(* Logix 5000 project; controller CarbonScout_MK6 vendor 1 type 14 code 154 rev 32.11; software revision 32.00; part 4 of 17 *)
(* tags used below, declared in another part *)
   Cfg_Exists : BOOL;   // 1=Alarm configured to exist, 0=Does not exist, don't scan
   Cfg_ResetReqd : BOOL;   // 1=Latched Alarm, a Reset is required to clear this Alarm
   Cfg_AckReqd : BOOL;   // 1=Acknowledge required for this Alarm
   Cfg_AllowShelve : BOOL;   // 1=Allow Operator to Shelve this Alarm
   Cfg_AllowDisable : BOOL;   // 1=Allow Maintenance to Disable this Alarm
   Cfg_Severity : DINT;   // Alarm Severity: 1..250=Low, 251..500=Medium, 501..750=High, 751..1000=Urgent
   Cfg_AlmMinOnT : DINT;   // Minimum time Alm output stays on (sec)
   PCfg_AllowExist : BOOL;   // 1=Alarm can be configured to exist, 0=other configs make alarm meaningless
   PCmd_Ack : BOOL;   // Program Command to Acknowledge alarm
   PCmd_Suppress : BOOL;   // Program Command to Suppress by Design (inhibits new alarm)
   PCmd_Unsuppress : BOOL;   // Program Command to Unsuppress (allows new alarm)
   PCmd_Unshelve : BOOL;   // Program Command to Unshelve (e.g., on shift change)
   OCmd_Ack : BOOL;   // Operator Command to Acknowledge alarm
   OCmd_Shelve : BOOL;   // Operator Command to Shelve Alarm (inhibits new alarm)
   OCmd_Unshelve : BOOL;   // Operator Command to Unshelve alarm (allows new alarm)
   Alm : ALIAS FOR Com_AE.0;   // Alarm output 1=In Alarm
   Ack : ALIAS FOR Com_AE.1;   // Alarm acknowledged status: 1=Ack rcvd
   Shelved : ALIAS FOR Com_AE.3;   // 1=Alarm has been Shelved by Operator (inhibits new alarm)
   Suppressed : ALIAS FOR Com_AE.6;   // 1=Alarm has been Suppressed by Program (inhibits new alarm)
   Disabled : ALIAS FOR Com_AE.9;   // 1=Alarm has been Disabled by Maintanance (inhibits new alarm)
   P_Alarm : BOOL;   // Unique Parameter Name for auto - discovery
   Wrk_Suppressed : BOOL;   // Internal Alarm Suppressed Status
   Com_AE : DINT;   // Communication with HMI / Alarm/Event Server (see bit descriptions)
   Simulation : DINT;
   test : DINT;
(* P_Alarm, continued *)

ROUTINE Prescan   (* ladder *)
// Clear "lurking" Commands
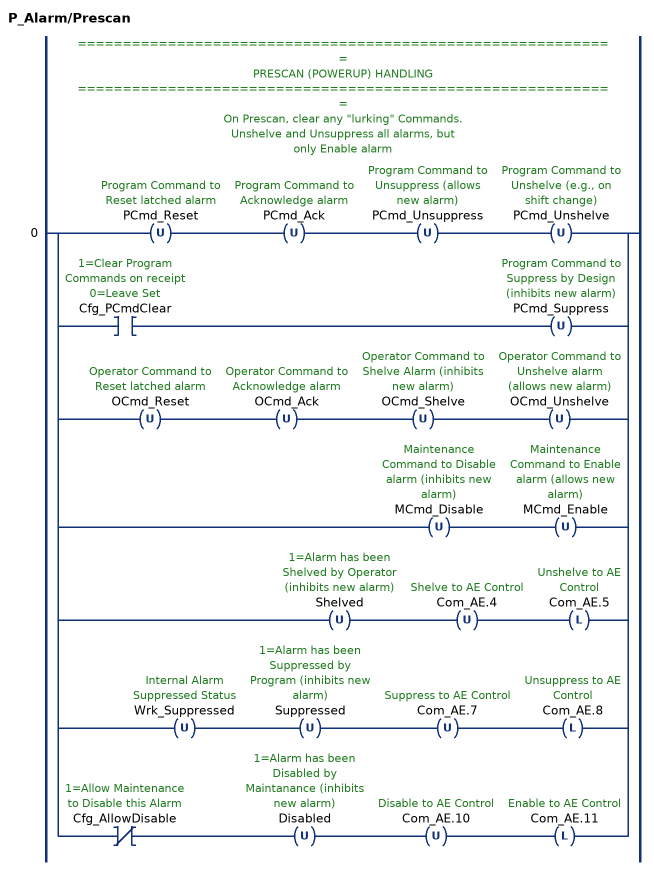
   // ============================================================
   // PRESCAN (POWERUP) HANDLING
   // ============================================================
   // On Prescan, clear any "lurking" Commands.
   // Unshelve and Unsuppress all alarms, but
   // only Enable alarm
   0: [OTU(PCmd_Reset) OTU(PCmd_Ack) OTU(PCmd_Unsuppress) OTU(PCmd_Unshelve) ,XIC(Cfg_PCmdClear) OTU(PCmd_Suppress) ,OTU(OCmd_Reset) OTU(OCmd_Ack) OTU(OCmd_Shelve) OTU(OCmd_Unshelve) ,OTU(MCmd_Disable) OTU(MCmd_Enable) ,OTU(Shelved) OTU(Com_AE.4) OTL(Com_AE.5) ,OTU(Wrk_Suppressed) OTU(Suppressed) OTU(Com_AE.7) OTL(Com_AE.8) ,XIO(Cfg_AllowDisable) OTU(Disabled) OTU(Com_AE.10) OTL(Com_AE.11) ];
END_ROUTINE
END_ADD_ON_INSTRUCTION

ADD_ON_INSTRUCTION P_Gate   (* revision 3.5 01 Release, vendor Rockwell Automation, ExecutePrescan, ExecuteEnableInFalse *)
// Condition Gate/Delay
// Revision note:
// See V3.5-xx Release Notes for details. Unchanged, up-rev only for V3.5 Library.
// Help:
// Copyright © Rockwell Automation, Inc.  All Rights Reserved.
// This Instruction provides a "gate" for a discrete Input signal and
// provides on-delay and off-delay timing for the gated signal.
// When the Gate input is true, the instruction Input is passed through
// to the Output, with on-delay and off-delay timing applied.
// When the Gate input is false, the Output is kept off
// (note: off-delay still applies!)
// This instruction is usually used between a comparison
// (analog threshold with deadband or discrete logic)
// and a P_Alarm instance, but may be used as a
// gated on-delay/off-delay timer generally.
// When EnableIn  is FALSE (e.g., on a false LD rung),
// the Input "Inp" is inverted.  Note that the Gate
// input (Inp_Gate) is NOT inverted!!!
VAR_INPUT
   Inp : BOOL; {visible}   // Input Condition: e.g., result of comparison
   Inp_Gate : BOOL := 1; {visible}   // Gate Input: 1=enable On Delay / Off Delay after Gate Delay, 0=disable
   Cfg_GateDly : DINT;   // Gate Delay (s): time after Gate Input true to enable On/Off Delay
   Cfg_OnDly : DINT;   // On Delay (s): If Gate Delay done, time Inp must be true to set Out true
   Cfg_OffDly : DINT;   // Off Delay (s): Time after Inp or Gate goes to 0 for Out to go to 0
END_VAR
VAR_OUTPUT
   Out : BOOL; {access Read Only, visible}   // Output after On Delay, Off Delay, enabled by Gate
   Sts_Gate : BOOL; {access Read Only, visible}   // 1=Gate Delay done, Output is enabled
   Sts_Err : BOOL; {access Read Only, visible}   // 1=Error in Config (see detail Err_ bits for reason), display icon
   Err_Timer : BOOL; {access Read Only}   // 1=Error in Config: On Delay, Off Delay, Gate Delay Time Invalid (use 0 to 2147483 s)
   P_Gate : BOOL;   // Unique Parameter Name for auto - discovery
END_VAR
VAR
   Wrk_OffDlyT : TIMER; {access Read Only}   // Off Delay Timer
   Wrk_OnDlyT : TIMER; {access Read Only}   // On Delay Timer
   Wrk_GateT : TIMER; {access Read Only}   // Gate Delay Timer
   Cfg_InpCond : STRING_8;   // Displayed text of P_Gate's Input (Inp) Condition
   Inf_Tab : DINT;   // Tab to display (FTView ME)
END_VAR

ROUTINE EnableInFalse   (* ladder *)
// Same as main Logic routine, except Inp is inverted (for use in LD logic)  (Inp_Gate is NOT inverted!!!)
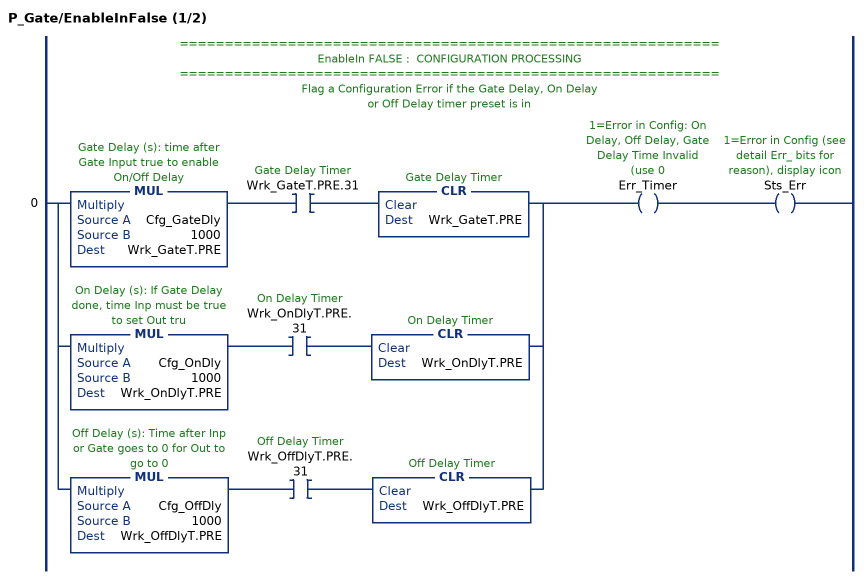
   // ============================================================
   // EnableIn FALSE :  CONFIGURATION PROCESSING
   // ============================================================
   // Flag a Configuration Error if the Gate Delay, On Delay
   // or Off Delay timer preset is in
   0: [MUL(Cfg_GateDly,1000,Wrk_GateT.PRE) XIC(Wrk_GateT.PRE.31) CLR(Wrk_GateT.PRE) ,MUL(Cfg_OnDly,1000,Wrk_OnDlyT.PRE) XIC(Wrk_OnDlyT.PRE.31) CLR(Wrk_OnDlyT.PRE) ,MUL(Cfg_OffDly,1000,Wrk_OffDlyT.PRE) XIC(Wrk_OffDlyT.PRE.31) CLR(Wrk_OffDlyT.PRE) ]OTE(Err_Timer)OTE(Sts_Err);
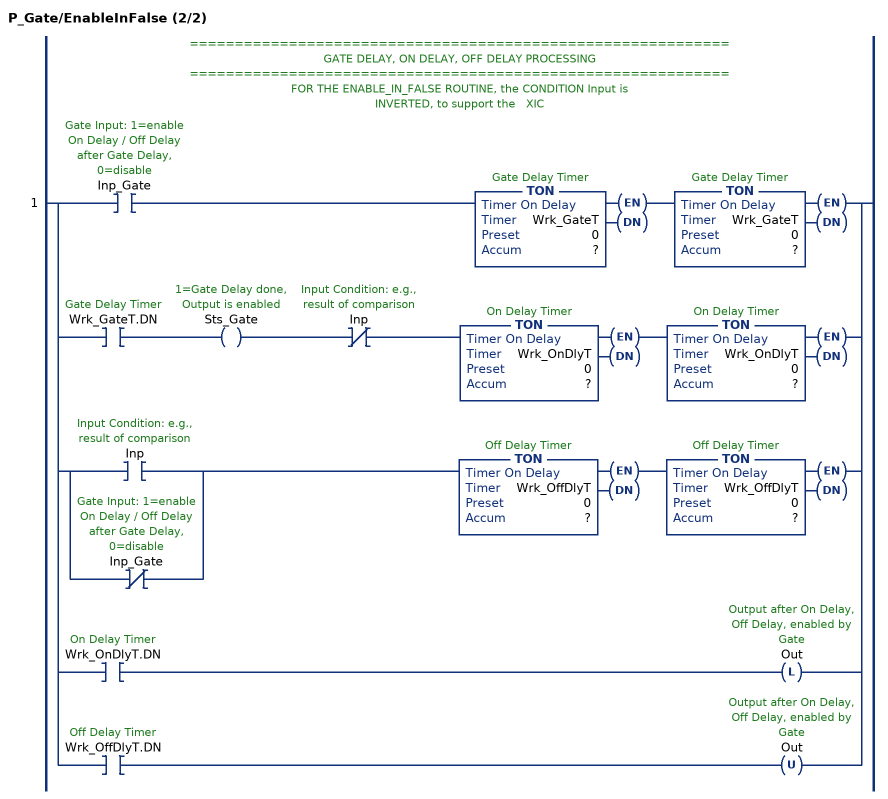
   // ============================================================
   // GATE DELAY, ON DELAY, OFF DELAY PROCESSING
   // ============================================================
   // FOR THE ENABLE_IN_FALSE ROUTINE, the CONDITION Input is
   // INVERTED, to support the   XIC
   1: [XIC(Inp_Gate) TON(Wrk_GateT,?,?) TON(Wrk_GateT,?,?) ,XIC(Wrk_GateT.DN) OTE(Sts_Gate) XIO(Inp) TON(Wrk_OnDlyT,?,?) TON(Wrk_OnDlyT,?,?) ,[XIC(Inp) ,XIO(Inp_Gate) ] TON(Wrk_OffDlyT,?,?) TON(Wrk_OffDlyT,?,?) ,XIC(Wrk_OnDlyT.DN) OTL(Out) ,XIC(Wrk_OffDlyT.DN) OTU(Out) ];
END_ROUTINE

ROUTINE Logic   (* ladder *)
// Gate the input and apply on-delay and off-delay timing
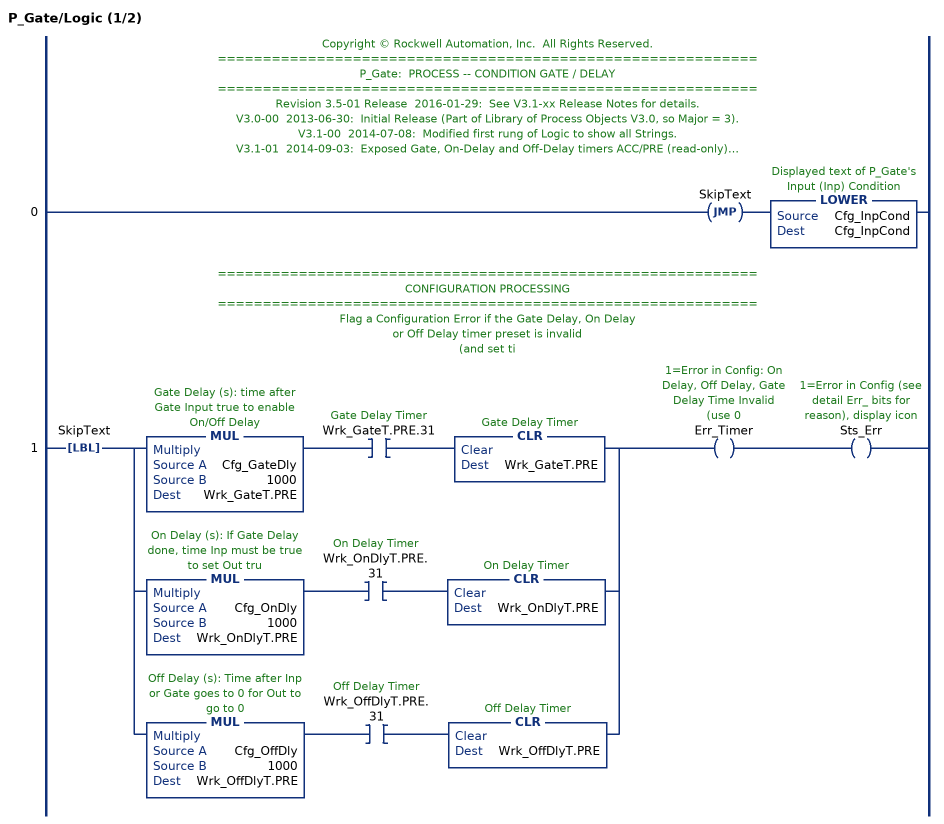
   // Copyright © Rockwell Automation, Inc.  All Rights Reserved.
   // ============================================================
   // P_Gate:  PROCESS -- CONDITION GATE / DELAY
   // ============================================================
   // Revision 3.5-01 Release  2016-01-29:  See V3.1-xx Release Notes for details.
   // V3.0-00  2013-06-30:  Initial Release (Part of Library of Process Objects V3.0, so Major = 3).
   // V3.1-00  2014-07-08:  Modified first rung of Logic to show all Strings.
   // V3.1-01  2014-09-03:  Exposed Gate, On-Delay and Off-Delay timers ACC/PRE (read-only).
   // V3.1-05  2016-01-22:  Corrected logic when using analog threshold with deadband.
   // V3.5-01  2016-01-29:  Unchanged, up-rev only for V3.5 Library.
   // ============================================================
   // This Instruction provides a "gate" for a discrete Input signal and
   // provides on-delay and off-delay timing for the gated signal.
   // When the Gate input is true, the instruction Input is passed through
   // to the Output, with on-delay and off-delay timing applied.
   // When the Gate input is false, the Output is kept off
   // (note: off-delay still applies!)
   // This instruction is usually used between a comparison
   // (analog threshold with deadband or discrete logic)
   // and a P_Alarm instance, but may be used as a
   // gated on-delay/off-delay timer generally.
   // When EnableIn  is FALSE (e.g., on a false LD rung),
   // the Input "Inp" is inverted.  Note that the Gate
   // input (Inp_Gate) is NOT inverted!!!
   // ============================================================
   // SHOW LOCAL STRINGS
   // ============================================================
   // The STRINGs containing the text associated with each instance of this
   // instruction cannot be Input or Output Parameters, because STRINGs are not
   //  'atomic' types. (Inputs and Outputs must be SINT, INT, DINT, REAL, or BOOL.)
   // In order to make it easier to find and configure these STRINGs, this rung
   // was added.  THE JMP (and the LBL on the following rung)
   // MUST NOT BE REMOVED!!!
   // To view the STRINGs, go to the instruction instance (in LD or FBD), RIGHT-click
   // to bring up the context menu and select "Open Instruction Logic".
   // This rung will appear with the STRING values for the selected instance.
   // You may double-click the STRING values here to modify them as well.
   // #####  V3.1-00  2014-07-08: Added Inf_Type to displayed Strings  #####
   0: JMP(SkipText)LOWER(Cfg_InpCond,Cfg_InpCond);
   // ============================================================
   // CONFIGURATION PROCESSING
   // ============================================================
   // Flag a Configuration Error if the Gate Delay, On Delay
   // or Off Delay timer preset is invalid
   // (and set ti
   1: LBL(SkipText)[MUL(Cfg_GateDly,1000,Wrk_GateT.PRE) XIC(Wrk_GateT.PRE.31) CLR(Wrk_GateT.PRE) ,MUL(Cfg_OnDly,1000,Wrk_OnDlyT.PRE) XIC(Wrk_OnDlyT.PRE.31) CLR(Wrk_OnDlyT.PRE) ,MUL(Cfg_OffDly,1000,Wrk_OffDlyT.PRE) XIC(Wrk_OffDlyT.PRE.31) CLR(Wrk_OffDlyT.PRE) ]OTE(Err_Timer)OTE(Sts_Err);
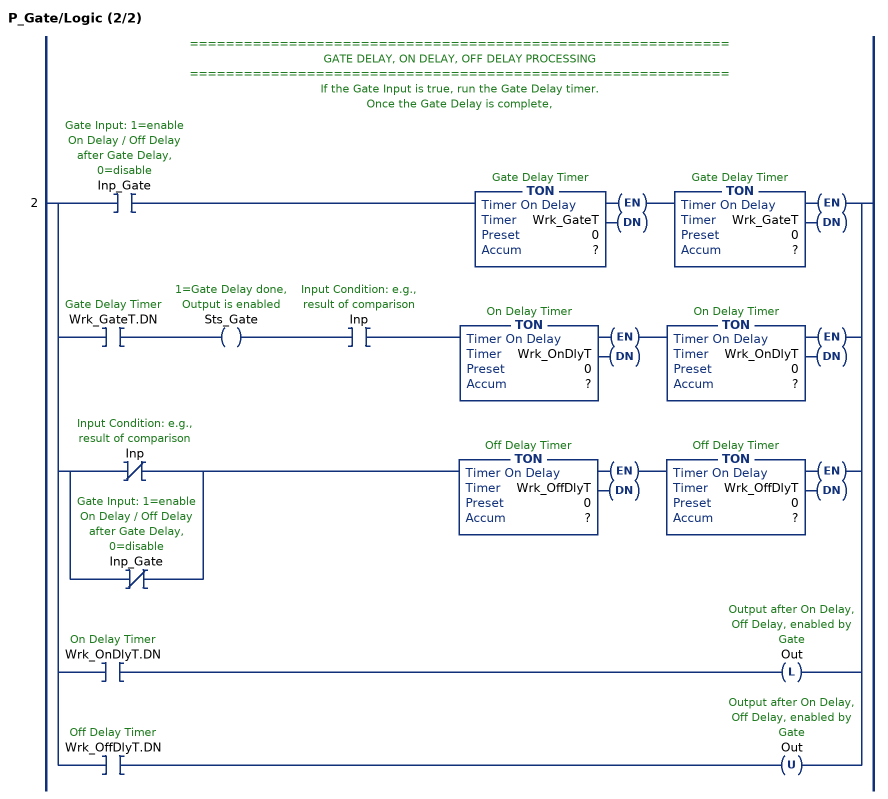
   // ============================================================
   // GATE DELAY, ON DELAY, OFF DELAY PROCESSING
   // ============================================================
   // If the Gate Input is true, run the Gate Delay timer.
   // Once the Gate Delay is complete,
   2: [XIC(Inp_Gate) TON(Wrk_GateT,?,?) TON(Wrk_GateT,?,?) ,XIC(Wrk_GateT.DN) OTE(Sts_Gate) XIC(Inp) TON(Wrk_OnDlyT,?,?) TON(Wrk_OnDlyT,?,?) ,[XIO(Inp) ,XIO(Inp_Gate) ] TON(Wrk_OffDlyT,?,?) TON(Wrk_OffDlyT,?,?) ,XIC(Wrk_OnDlyT.DN) OTL(Out) ,XIC(Wrk_OffDlyT.DN) OTU(Out) ];
END_ROUTINE

ROUTINE Prescan   (* ladder *)
// Set the Gate Input to 1 (default value) on prescan
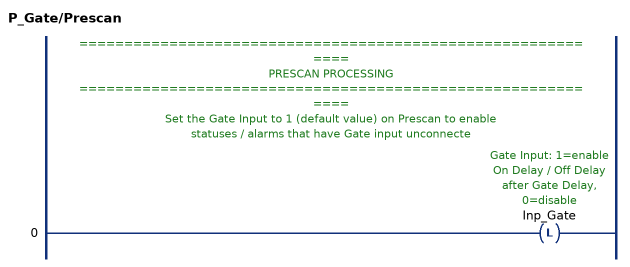
   // ============================================================
   // PRESCAN PROCESSING
   // ============================================================
   // Set the Gate Input to 1 (default value) on Prescan to enable
   // statuses / alarms that have Gate input unconnecte
   0: OTL(Inp_Gate);
END_ROUTINE
END_ADD_ON_INSTRUCTION

ADD_ON_INSTRUCTION P_Mode   (* revision 3.5 01 Release, vendor Rockwell Automation, ExecutePrescan, ExecuteEnableInFalse *)
// Mode
// Revision note:
// See V3.5-xx Release Notes for details. Unmodified, up-rev only for V3.5-01 Release.
// Help:
// Copyright © Rockwell Automation, Inc.  All Rights Reserved.
// This instruction provides selection of Mode (owner) for a Device level
// object  (from highest priority to lowest):
// *  No Mode (no owner, EnableIn is false)
// *  Hand (typically tracks hardwired control of device)
// *  Maint (Maintenance) (taken out of normal service for maintenance)
// *  Ovrd (Override) (typically used for process overrides)
// *  Prog  (Program) (automated control, and default if Cfg_ProgNorm = 1)
// *  Oper (Operator (manual control, and default if Cfg_ProgNorm = 0)
// (Program and Operator have the same priority.)
// The current mode is shown with Status bits and also as the primary
// Value for the instruction: an enumeration "Val" as follows:
//   0 = No Mode,
//   1 = Hand,
//   2 = Maintenance,
//   3 = Override,
//   4 = Program (Locked),
//   5 = Operator (Locked),
//   6 = Program (Unlocked, Oper default),
//   7 = Operator (Unlocked, Prog default),
//   8 = Program (Unlocked, = default),
//   9 = Operator (Unlocked, = default).
// When EnableIn is false, all ownership acquire/release and lock/unlock
// Commands are processed "behind the scenes", but the Mode is shown
// as "No Mode" (no owner).  When EnableIn becomes true, the Mode
// takes into account the Commands received -- in other words, the Mode
// becomes the one that would have been in effect had the EnableIn
// False / No Mode condition never occurred.
VAR_INPUT
   Inp_Hand : BOOL; {visible}   // 1=Acquire Hand (typ. hardwired local) Mode, 0=Release Hand Mode
   Inp_Ovrd : BOOL; {visible}   // 1=Acquire Override (higher priority program logic) Mode, 0=Release Override Mode
   Cfg_PCmdClear : BOOL := 1;   // 1=Clear Program Command on receipt; 0=Use Level-based (maintained) PCmds
   Cfg_OvrdOverLock : BOOL := 1;   // 1=Override supersedes Prog/Oper Lock, 0=don't override Lock
   Cfg_ProgDefault : BOOL;   // Default Mode: 1=Program Mode if no requests; 0=Operator Mode if no requests
   PCmd_Acq : BOOL;   // Program Command to Acquire Ownership (Oper to Prog)
   PCmd_Rel : BOOL;   // Program Command to Release Ownership (Prog to Oper)
   PCmd_Lock : BOOL;   // Program Command to Lock Mode in Prog
   PCmd_Unlock : BOOL;   // Program Command to Unlock Mode
   MCmd_Acq : BOOL;   // Maintenance Command to Acquire Ownership (Oper/Prog/Ovrd to Maint)
   MCmd_Rel : BOOL;   // Maintenance Command to Release Ownership (Maint to Oper/Prog/Ovrd)
   OCmd_AcqLock : BOOL;   // Operator Command to Acquire (Prog to Oper) / Lock Ownership
   OCmd_UnlockRel : BOOL;   // Operator Command to Unlock / Release (Oper to Prog) Ownership
END_VAR
VAR_OUTPUT
   Val : DINT; {access Read Only}   // Mode enum: 0=No, 1=H, 2=M, 3=!, 4=P Lock, 5=O Lock, 6=P (O Def), 7=O (P Def), 8=P (= Def), 9=O (= Def)
   Sts_Hand : BOOL; {access Read Only, visible}   // 1=Mode is Hand (supersedes Maint, Ovrd, Prog, Oper)
   Sts_Maint : BOOL; {access Read Only, visible}   // 1=Mode is Maintenance (supersedes Ovrd, Prog, Oper)
   Sts_Ovrd : BOOL; {access Read Only, visible}   // 1=Mode is Override (supersedes Prog, Oper)
   Sts_Prog : BOOL; {access Read Only, visible}   // 1=Mode is Program
   Sts_Oper : BOOL := 1; {access Read Only, visible}   // 1=Mode is Operator
   Sts_ProgOperLock : BOOL; {access Read Only, visible}   // 1=Program or Operator has requested Mode Lock
   Sts_ProgOperSel : BOOL; {access Read Only}   // Prog/Oper selection 1=Program, 0=Operator
   Sts_NoMode : BOOL; {access Read Only}   // 1=Mode is No Mode (no owner, disabled or not scanned)
   Sts_MAcqRcvd : BOOL; {access Read Only}   // 1=Maintenance Acquire command received this scan
   Rdy_MAcq : BOOL; {access Read Only}   // 1=Ready for MCmd_Acq, enable button
   Rdy_MRel : BOOL; {access Read Only}   // 1=Ready for MCmd_Rel, enable button
   Rdy_OAcq : BOOL; {access Read Only}   // 1=Ready for OCmd_AcqLock, enable Acquire (to Oper) button
   Rdy_OLock : BOOL; {access Read Only}   // 1=Ready for OCmd_AcqLock, enable Oper Lock button
   Rdy_OUnlock : BOOL; {access Read Only}   // 1=Ready for OCmd_UnlockRel, enable Oper Unlock button
   Rdy_ORel : BOOL; {access Read Only}   // 1=Ready for OCmd_UnlockRel, enable Release (to Prog) button
   P_Mode : BOOL;   // Unique Parameter Name for auto - discovery
END_VAR
VAR
   Wrk_Locked : BOOL; {access None}   // 1=Program/Operator Mode selection is Locked
   Wrk_Prog : BOOL; {access None}   // Internal Program (1) / Operator (0) Mode selection
   Wrk_Maint : BOOL; {access None}   // Internal Maintenance Mode
END_VAR

ROUTINE EnableInFalse   (* ladder *)
// Processes received Commands, but shows "NO mode" (no owner)
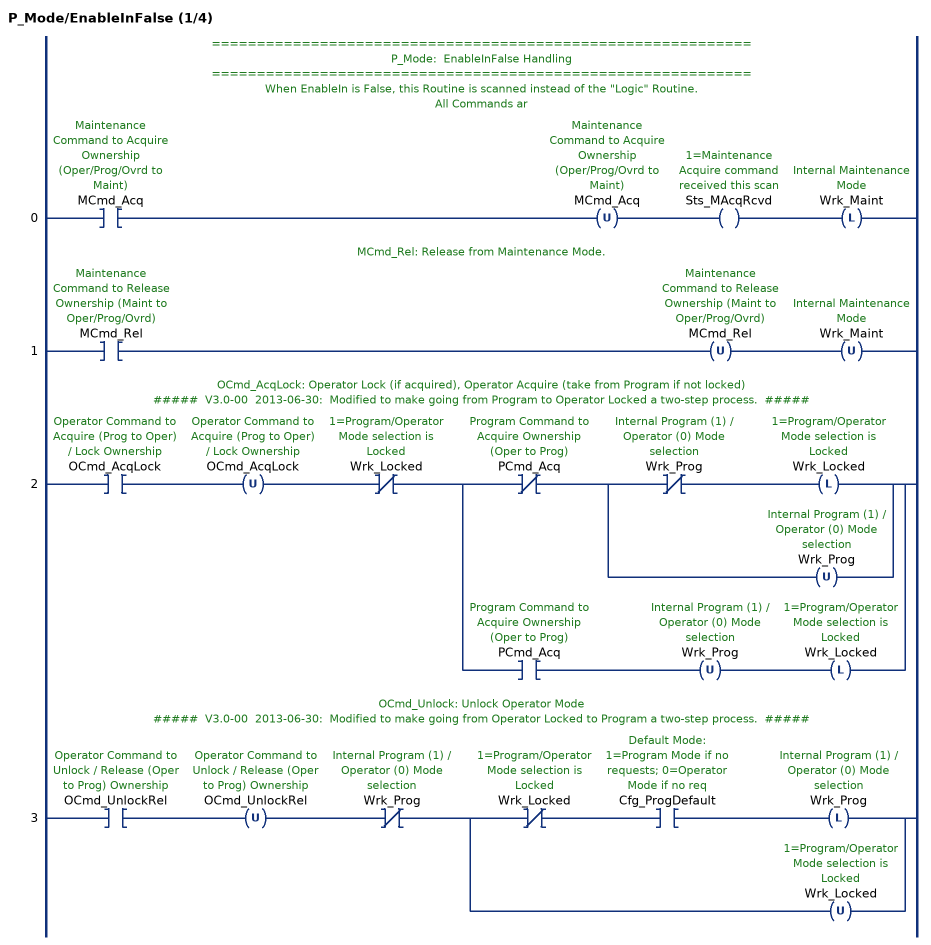
   // ============================================================
   // P_Mode:  EnableInFalse Handling
   // ============================================================
   // When EnableIn is False, this Routine is scanned instead of the "Logic" Routine.
   // All Commands ar
   0: XIC(MCmd_Acq)OTU(MCmd_Acq)OTE(Sts_MAcqRcvd)OTL(Wrk_Maint);
   // MCmd_Rel: Release from Maintenance Mode.
   1: XIC(MCmd_Rel)OTU(MCmd_Rel)OTU(Wrk_Maint);
   // OCmd_AcqLock: Operator Lock (if acquired), Operator Acquire (take from Program if not locked)
   // #####  V3.0-00  2013-06-30:  Modified to make going from Program to Operator Locked a two-step process.  #####
   2: XIC(OCmd_AcqLock)OTU(OCmd_AcqLock)XIO(Wrk_Locked)[XIO(PCmd_Acq) [XIO(Wrk_Prog) OTL(Wrk_Locked) ,OTU(Wrk_Prog) ] ,XIC(PCmd_Acq) OTU(Wrk_Prog) OTL(Wrk_Locked) ];
   // OCmd_Unlock: Unlock Operator Mode
   // #####  V3.0-00  2013-06-30:  Modified to make going from Operator Locked to Program a two-step process.  #####
   3: XIC(OCmd_UnlockRel)OTU(OCmd_UnlockRel)XIO(Wrk_Prog)[XIO(Wrk_Locked) XIC(Cfg_ProgDefault) OTL(Wrk_Prog) ,OTU(Wrk_Locked) ];
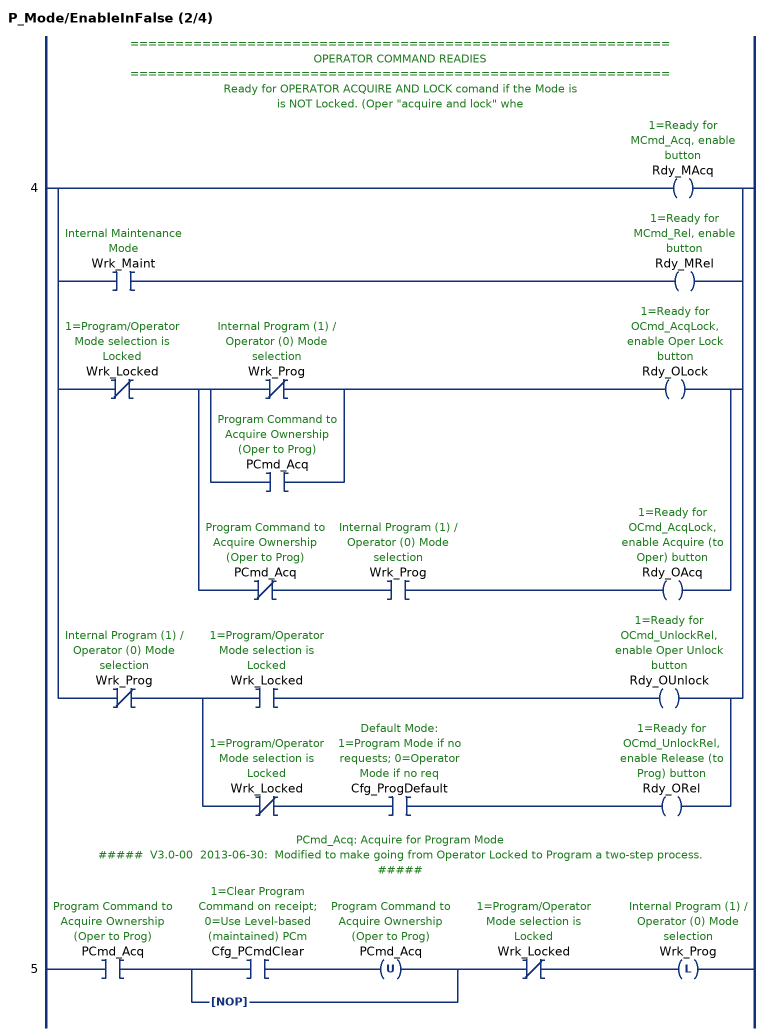
   // ============================================================
   // OPERATOR COMMAND READIES
   // ============================================================
   // Ready for OPERATOR ACQUIRE AND LOCK comand if the Mode is
   //  is NOT Locked. (Oper "acquire and lock" whe
   4: [OTE(Rdy_MAcq) ,XIC(Wrk_Maint) OTE(Rdy_MRel) ,XIO(Wrk_Locked) [[XIO(Wrk_Prog) ,XIC(PCmd_Acq) ] OTE(Rdy_OLock) ,XIO(PCmd_Acq) XIC(Wrk_Prog) OTE(Rdy_OAcq) ] ,XIO(Wrk_Prog) [XIC(Wrk_Locked) OTE(Rdy_OUnlock) ,XIO(Wrk_Locked) XIC(Cfg_ProgDefault) OTE(Rdy_ORel) ] ];
   // PCmd_Acq: Acquire for Program Mode
   // #####  V3.0-00  2013-06-30:  Modified to make going from Operator Locked to Program a two-step process.  #####
   5: XIC(PCmd_Acq)[XIC(Cfg_PCmdClear) OTU(PCmd_Acq) ,NOP() ]XIO(Wrk_Locked)OTL(Wrk_Prog);
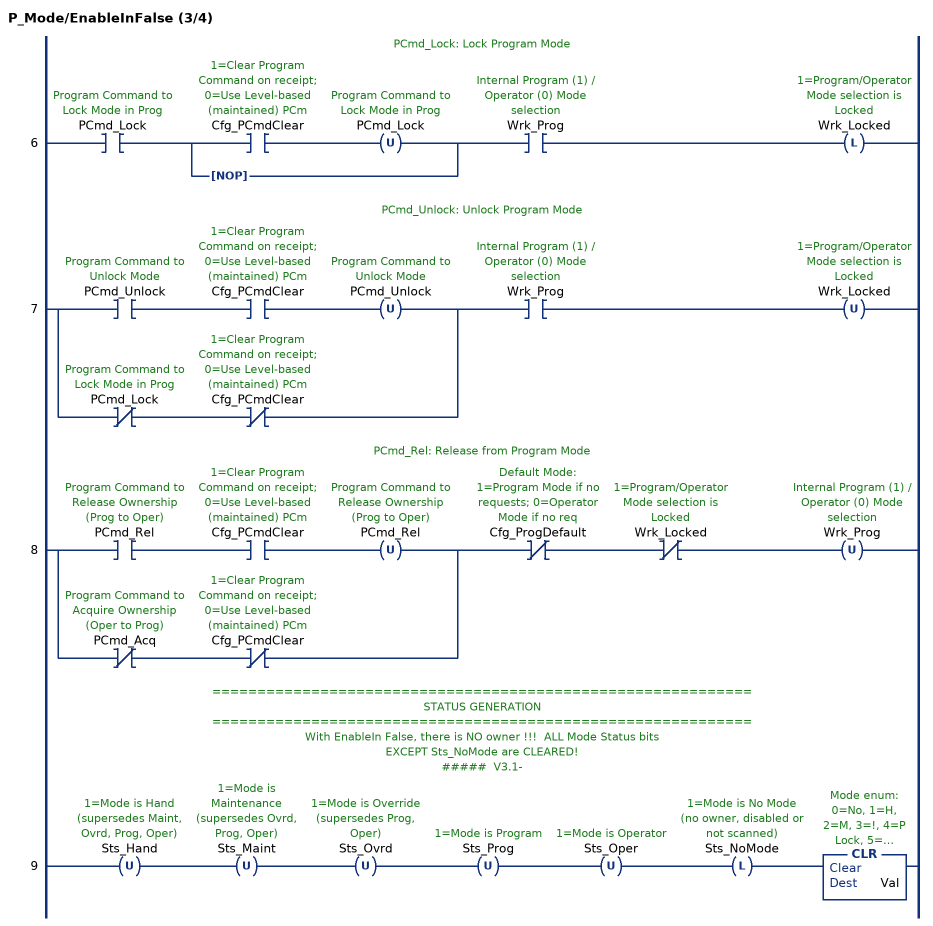
   // PCmd_Lock: Lock Program Mode
   6: XIC(PCmd_Lock)[XIC(Cfg_PCmdClear) OTU(PCmd_Lock) ,NOP() ]XIC(Wrk_Prog)OTL(Wrk_Locked);
   // PCmd_Unlock: Unlock Program Mode
   7: [XIC(PCmd_Unlock) XIC(Cfg_PCmdClear) OTU(PCmd_Unlock) ,XIO(PCmd_Lock) XIO(Cfg_PCmdClear) ]XIC(Wrk_Prog)OTU(Wrk_Locked);
   // PCmd_Rel: Release from Program Mode
   8: [XIC(PCmd_Rel) XIC(Cfg_PCmdClear) OTU(PCmd_Rel) ,XIO(PCmd_Acq) XIO(Cfg_PCmdClear) ]XIO(Cfg_ProgDefault)XIO(Wrk_Locked)OTU(Wrk_Prog);
   // ============================================================
   // STATUS GENERATION
   // ============================================================
   // With EnableIn False, there is NO owner !!!  ALL Mode Status bits
   // EXCEPT Sts_NoMode are CLEARED!
   // #####  V3.1-
   9: OTU(Sts_Hand)OTU(Sts_Maint)OTU(Sts_Ovrd)OTU(Sts_Prog)OTU(Sts_Oper)OTL(Sts_NoMode)CLR(Val);
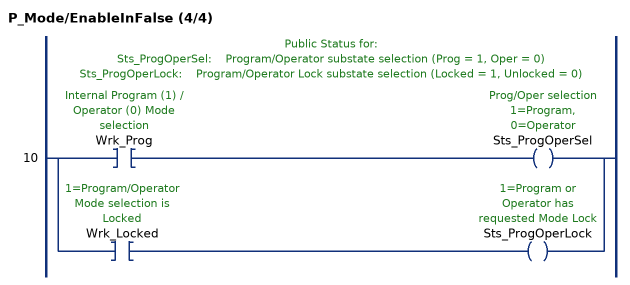
   // Public Status for:
   // Sts_ProgOperSel:    Program/Operator substate selection (Prog = 1, Oper = 0)
   // Sts_ProgOperLock:    Program/Operator Lock substate selection (Locked = 1, Unlocked = 0)
   10: [XIC(Wrk_Prog) OTE(Sts_ProgOperSel) ,XIC(Wrk_Locked) OTE(Sts_ProgOperLock) ];
END_ROUTINE

ROUTINE Logic   (* ladder *)
// Selects Modes (Hand, Maint, Ovrd, Oper, Prog) based on Inputs and Commands
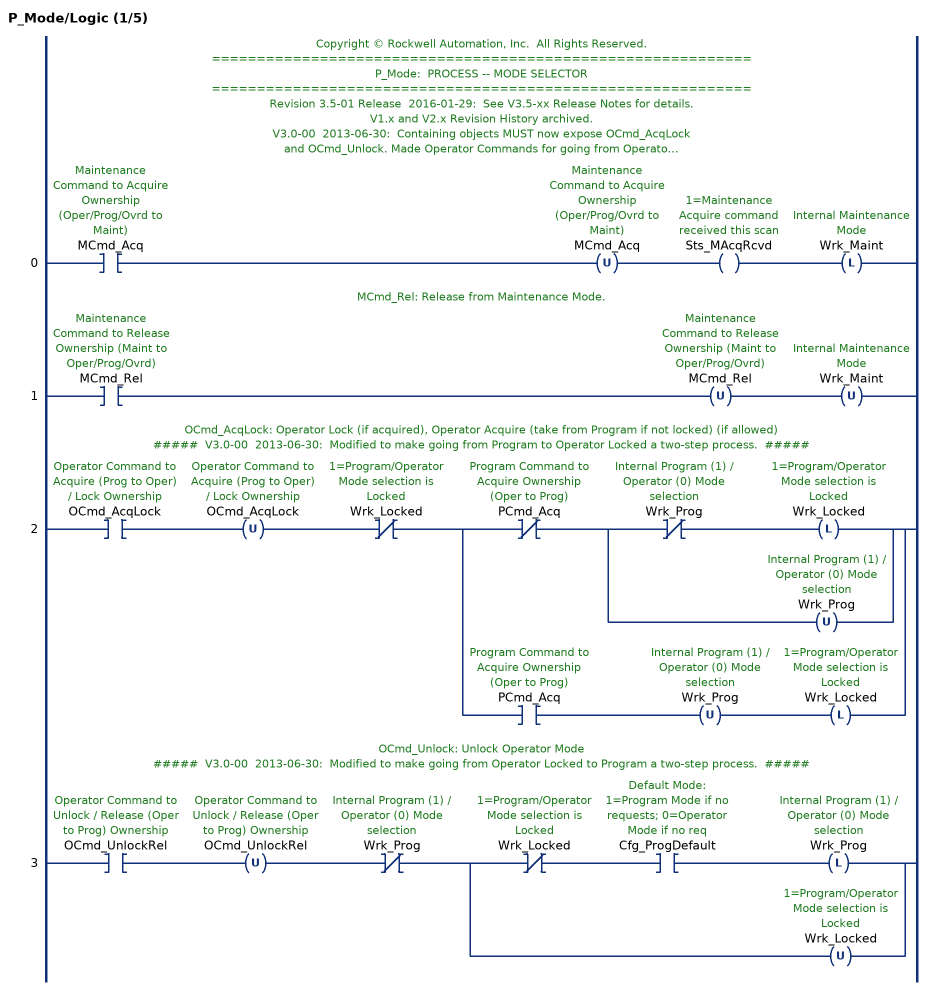
   // Copyright © Rockwell Automation, Inc.  All Rights Reserved.
   // ============================================================
   // P_Mode:  PROCESS -- MODE SELECTOR
   // ============================================================
   // Revision 3.5-01 Release  2016-01-29:  See V3.5-xx Release Notes for details.
   // V1.x and V2.x Revision History archived.
   // V3.0-00  2013-06-30:  Containing objects MUST now expose OCmd_AcqLock
   // and OCmd_Unlock. Made Operator Commands for going from Operator
   // Locked to Program (unlocked) and Program (unlocked) to Operator
   // Lock two-step processes.  Added Inf_Lib, Inf_Type.
   // V3.1-00  2014-06-30:  Containing objects must expose Maintenance Acquire /
   // Release commands and new Sts_MAcqRcvd.
   // Changed Val (enum) to SINT. Fixed parameter descriptions.
   // V3.1-01  2014-09-03:  Unmodified, up-rev only for V3.1-01 public release.
   // V3.5-01  2016-01-29:  Unmodified, up-rev only for V3.5-01 Release.
   // ============================================================
   // This instruction provides selection of Mode (owner) for a Device level
   // object  (from highest priority to lowest):
   // * NO Mode (EnableIn is false)
   // *  Hand (typically tracks hardwired control of device)
   // *  Maint (Maintenance) (taken out of normal service for maintenance)
   // *  Ovrd (Override) (typically used for process overrides)
   // *  Prog  (Program) (automated control, and default if Cfg_ProgNorm = 1)
   // *  Oper (Operator (manual control, and default if Cfg_ProgNorm = 0)
   // The current mode is shown with Status bits and also as the
   // primary Value for the instruction: an enumeration as follows:
   // 0 = No Mode, 1 = Hand, 2 = Maintenance, 3 = Override,
   // 4 = Program (Locked), 5 = Operator (Locked),
   // 6 = Program (Unlocked, Oper default), 7 = Operator (Unlocked, Prog default),
   // 8 = Program (Unlocked, Prog default), 9 = Operator (Unlocked, Oper default).
   // ============================================================
   // COMMAND HANDLING
   // ============================================================
   // NOTE:  These rungs MUST be in the order given to meet the following
   // multiple-actions-at-the-same-time scenarios:
   // * Maintenance Release beats Maintenance Acquire
   // * Program Release beats Program Acquire
   // * Program Unlock beats Program Lock
   // * Operator Unlock beats Operator Acquire / Lock (results in Oper Unlocked)
   // * Program Acquire must come after Operator Unlock
   // If Cfg_ProgDefault = 1, the Mode defaults to Program
   // (instead of Operator) if all other Modes release their requests.
   // ============================================================
   // MCmd_Acq: Acquire for Maintenance Mode, and blink the status
   // that indicates a Maintenance Acquire command was received.
   // #####  V3.1-00  2014-06-30:  Added Sts_MAcqRcvd  #####
   0: XIC(MCmd_Acq)OTU(MCmd_Acq)OTE(Sts_MAcqRcvd)OTL(Wrk_Maint);
   // MCmd_Rel: Release from Maintenance Mode.
   1: XIC(MCmd_Rel)OTU(MCmd_Rel)OTU(Wrk_Maint);
   // OCmd_AcqLock: Operator Lock (if acquired), Operator Acquire (take from Program if not locked) (if allowed)
   // #####  V3.0-00  2013-06-30:  Modified to make going from Program to Operator Locked a two-step process.  #####
   2: XIC(OCmd_AcqLock)OTU(OCmd_AcqLock)XIO(Wrk_Locked)[XIO(PCmd_Acq) [XIO(Wrk_Prog) OTL(Wrk_Locked) ,OTU(Wrk_Prog) ] ,XIC(PCmd_Acq) OTU(Wrk_Prog) OTL(Wrk_Locked) ];
   // OCmd_Unlock: Unlock Operator Mode
   // #####  V3.0-00  2013-06-30:  Modified to make going from Operator Locked to Program a two-step process.  #####
   3: XIC(OCmd_UnlockRel)OTU(OCmd_UnlockRel)XIO(Wrk_Prog)[XIO(Wrk_Locked) XIC(Cfg_ProgDefault) OTL(Wrk_Prog) ,OTU(Wrk_Locked) ];
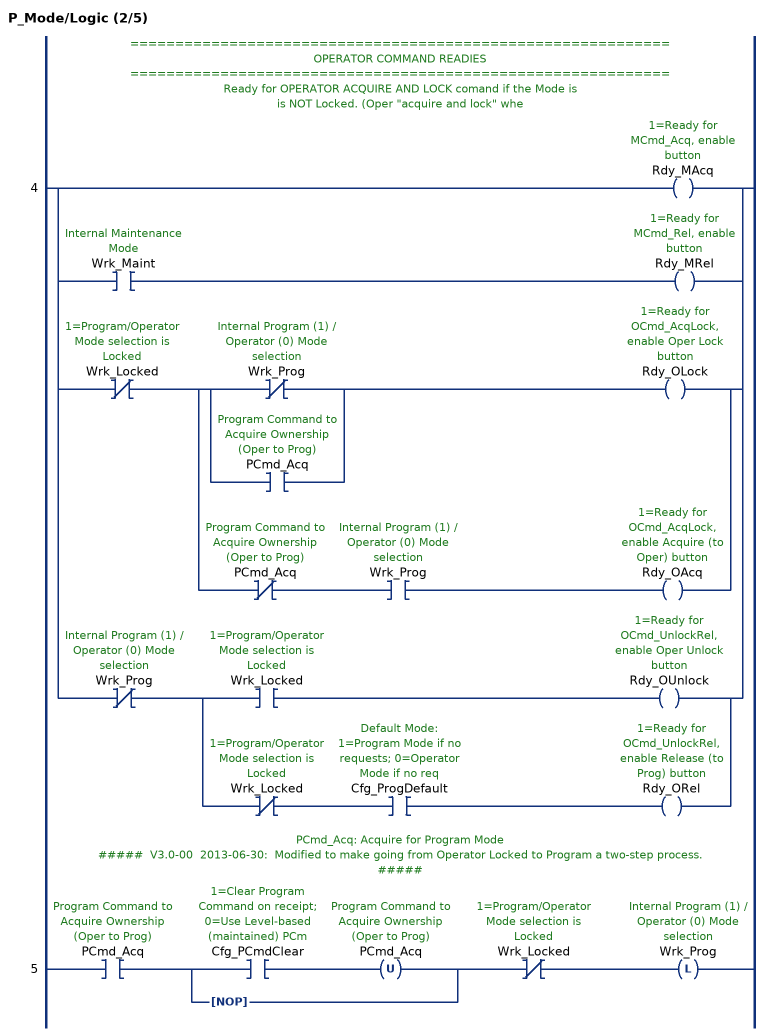
   // ============================================================
   // OPERATOR COMMAND READIES
   // ============================================================
   // Ready for OPERATOR ACQUIRE AND LOCK comand if the Mode is
   //  is NOT Locked. (Oper "acquire and lock" whe
   4: [OTE(Rdy_MAcq) ,XIC(Wrk_Maint) OTE(Rdy_MRel) ,XIO(Wrk_Locked) [[XIO(Wrk_Prog) ,XIC(PCmd_Acq) ] OTE(Rdy_OLock) ,XIO(PCmd_Acq) XIC(Wrk_Prog) OTE(Rdy_OAcq) ] ,XIO(Wrk_Prog) [XIC(Wrk_Locked) OTE(Rdy_OUnlock) ,XIO(Wrk_Locked) XIC(Cfg_ProgDefault) OTE(Rdy_ORel) ] ];
   // PCmd_Acq: Acquire for Program Mode
   // #####  V3.0-00  2013-06-30:  Modified to make going from Operator Locked to Program a two-step process.  #####
   5: XIC(PCmd_Acq)[XIC(Cfg_PCmdClear) OTU(PCmd_Acq) ,NOP() ]XIO(Wrk_Locked)OTL(Wrk_Prog);
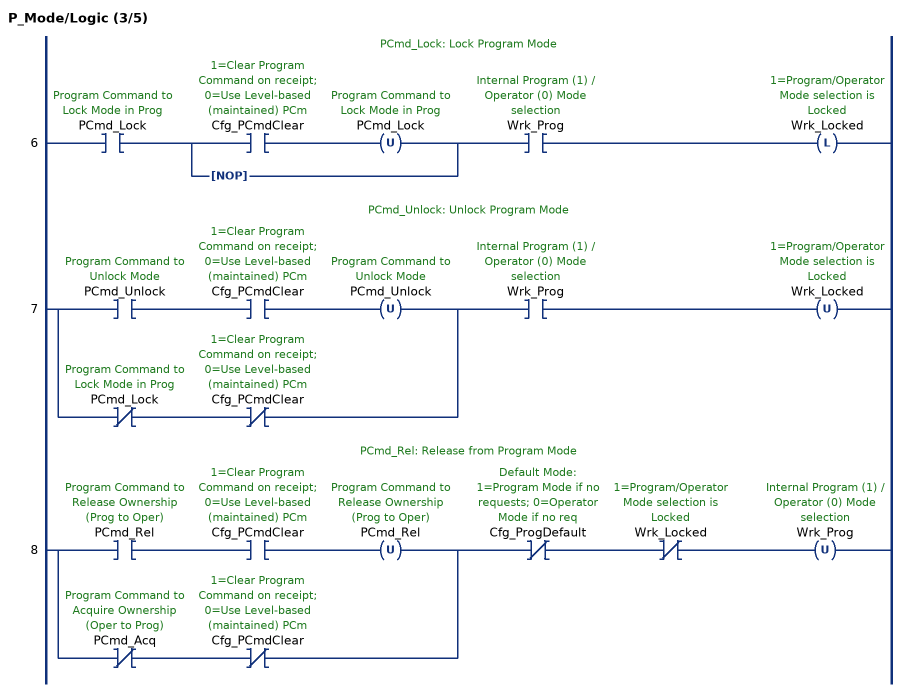
   // PCmd_Lock: Lock Program Mode
   6: XIC(PCmd_Lock)[XIC(Cfg_PCmdClear) OTU(PCmd_Lock) ,NOP() ]XIC(Wrk_Prog)OTL(Wrk_Locked);
   // PCmd_Unlock: Unlock Program Mode
   7: [XIC(PCmd_Unlock) XIC(Cfg_PCmdClear) OTU(PCmd_Unlock) ,XIO(PCmd_Lock) XIO(Cfg_PCmdClear) ]XIC(Wrk_Prog)OTU(Wrk_Locked);
   // PCmd_Rel: Release from Program Mode
   8: [XIC(PCmd_Rel) XIC(Cfg_PCmdClear) OTU(PCmd_Rel) ,XIO(PCmd_Acq) XIO(Cfg_PCmdClear) ]XIO(Cfg_ProgDefault)XIO(Wrk_Locked)OTU(Wrk_Prog);
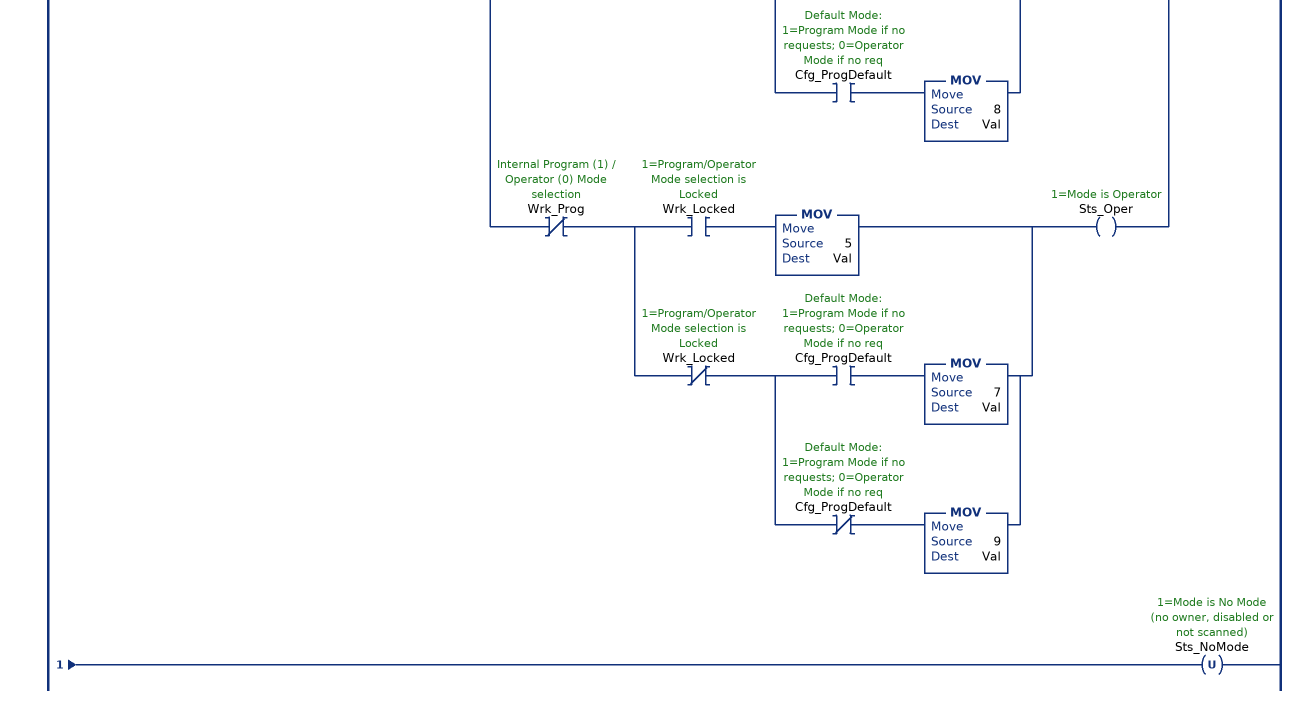
   // ============================================================
   // STATUS GENERATION
   // ============================================================
   // This rung determines the Mode based on the states of the inputs and internal working bits.
   // The logic here does
   9: [XIC(Inp_Hand) OTE(Sts_Hand) MOV(1,Val) ,XIO(Inp_Hand) [XIC(Wrk_Maint) OTE(Sts_Maint) MOV(2,Val) ,XIO(Wrk_Maint) [XIC(Inp_Ovrd) [XIO(Wrk_Locked) ,XIC(Cfg_OvrdOverLock) ,XIC(Sts_Ovrd) ] OTE(Sts_Ovrd) MOV(3,Val) ,XIO(Sts_Ovrd) [XIC(Wrk_Prog) [XIC(Wrk_Locked) MOV(4,Val) ,XIO(Wrk_Locked) [XIO(Cfg_ProgDefault) MOV(6,Val) ,XIC(Cfg_ProgDefault) MOV(8,Val) ] ] OTE(Sts_Prog) ,XIO(Wrk_Prog) [XIC(Wrk_Locked) MOV(5,Val) ,XIO(Wrk_Locked) [XIC(Cfg_ProgDefault) MOV(7,Val) ,XIO(Cfg_ProgDefault) MOV(9,Val) ] ] OTE(Sts_Oper) ] ] ] ]OTU(Sts_NoMode);
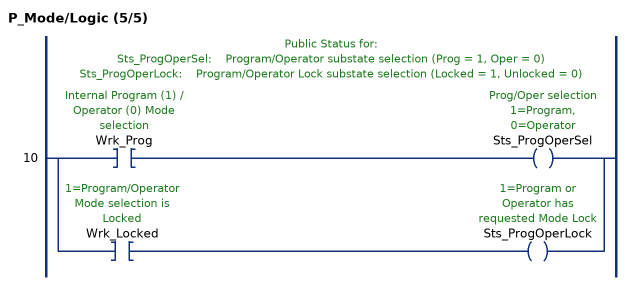
   // Public Status for:
   // Sts_ProgOperSel:    Program/Operator substate selection (Prog = 1, Oper = 0)
   // Sts_ProgOperLock:    Program/Operator Lock substate selection (Locked = 1, Unlocked = 0)
   10: [XIC(Wrk_Prog) OTE(Sts_ProgOperSel) ,XIC(Wrk_Locked) OTE(Sts_ProgOperLock) ];
END_ROUTINE

ROUTINE Prescan   (* ladder *)
// Clear "lurking" Commands
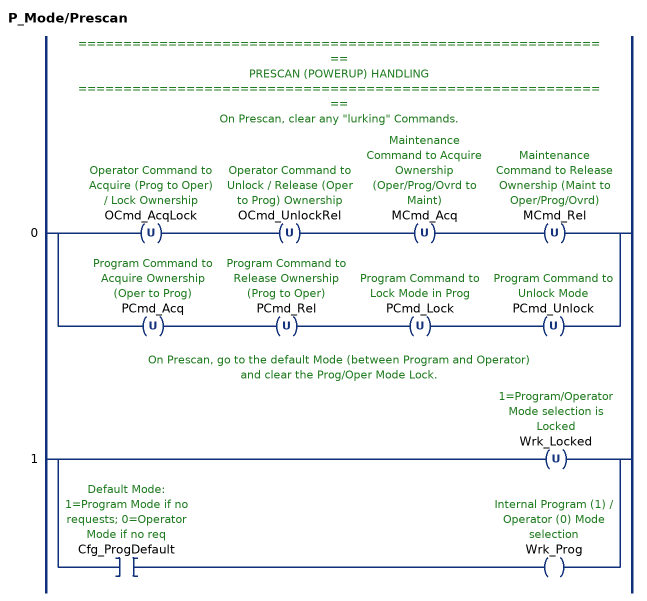
   // ============================================================
   // PRESCAN (POWERUP) HANDLING
   // ============================================================
   // On Prescan, clear any "lurking" Commands.
   0: [OTU(OCmd_AcqLock) OTU(OCmd_UnlockRel) OTU(MCmd_Acq) OTU(MCmd_Rel) ,OTU(PCmd_Acq) OTU(PCmd_Rel) OTU(PCmd_Lock) OTU(PCmd_Unlock) ];
   // On Prescan, go to the default Mode (between Program and Operator)
   // and clear the Prog/Oper Mode Lock.
   1: [OTU(Wrk_Locked) ,XIC(Cfg_ProgDefault) OTE(Wrk_Prog) ];
END_ROUTINE
END_ADD_ON_INSTRUCTION

ADD_ON_INSTRUCTION P_ValveSO   (* revision 3.5 04 Release, vendor Rockwell Automation, ExecutePrescan, ExecuteEnableInFalse *)
// Solenoid Operated Valve
// Revision note:
// See V3.5-xx Release Notes for details. Modified to align
// with actual device state on transition from Sim to real valve.
// Help:
// Copyright © Rockwell Automation, Inc.  All Rights Reserved.
// This Instruction controls and monitors a single solenoid operated
// valve (two position: opened, closed) and provides:
// *  Support for fail open (energize to close) and fail closed (energize to open, default) valves
// *  Monitoring of limit switch feedback, display of actual valve status
// *  Detection of Failure to Open, Failure to Close
// *  Monitoring of Permissive conditions to allow energizing
// *  Monitoring of Interlock conditions to de-energize
// *  Simulation, providing feedback of a working valve while disabling outputs
// *  Monitoring of I/O communication faults
// *  Alarms for Full Stall (didn't move), Transit Stall (didn't reach target position), Interlock Trip, I/O Fault
// *  Operation in Hand, Maintenance, Override, Program and Operator Modes
// *  "Available" status for use by automation logic to know whether valve
//       can be controlled by other objects.
// Modes are provided by a P_Mode AOI instance.
// Alarms are provided by P_Alarm AOI instances.
// Modes of operation: Operator, Program, Override, Maintenance, Hand
VAR_INPUT
   Inp_OpenLS : BOOL; {visible}   // Valve Open Limit Switch 1=confirmed OPEN
   Inp_ClosedLS : BOOL; {visible}   // Valve Closed Limit Switch 1=confirmed CLOSED
   Inp_PermOK : BOOL := 1; {visible}   // 1=Permissives OK, Valve can energize
   Inp_NBPermOK : BOOL := 1; {visible}   // 1=Non-Bypassable Permissives OK, valve can energize
   Inp_IntlkOK : BOOL := 1; {visible}   // 1=Interlocks OK, valve can energize
   Inp_NBIntlkOK : BOOL := 1; {visible}   // 1=Non-Bypassable Interlocks OK, valve can energize
   Inp_IOFault : BOOL; {visible}   // Input Communication Status 0=OK, 1=fail
   Inp_Sim : BOOL;   // 1=Simulate working valve; 0=Open/Close/ Monitor actual valve
   Inp_Hand : ALIAS FOR Mode.Inp_Hand; {visible}
   Inp_Ovrd : ALIAS FOR Mode.Inp_Ovrd; {visible}
   Inp_OvrdCmd : DINT; {visible}   // Override Mode Command: 0=None, 1=Close, 2=Open
   Inp_Reset : BOOL; {visible}   // 1=Reset all fault conditions and latched Alarms
   Cfg_FailOpen : BOOL;   // 1=Fail Open (energize to close), 0=Fail Closed (energize to open)
   Cfg_HasOpenLS : BOOL;   // 1=Valve provides an Open Limit Switch signal
   Cfg_HasClosedLS : BOOL;   // 1=Valve provides a Closed Limit Switch signal
   Cfg_UseOpenLS : BOOL;   // 1=Valve Open LS should be used for failure checking
   Cfg_UseClosedLS : BOOL;   // 1=Valve Closed LS should be used for failure checking
   Cfg_LSFail : BOOL := 1;   // 1=both switches ON=fail, 0=both switches OFF=fail
   Cfg_HasPermObj : BOOL;   // 1=Tells HMI a P_Perm is connected to Inp_Perm
   Cfg_HasIntlkObj : BOOL;   // 1=Tells HMI a P_Intlk is connected to Inp_Intlk
   Cfg_HasStatsObj : BOOL;   // 1=Tells HMI a P_ValveStats is monitoring this valve
   Cfg_PCmdClear : ALIAS FOR Mode.Cfg_PCmdClear;
   Cfg_ProgDefault : ALIAS FOR Mode.Cfg_ProgDefault;
   Cfg_OCmdResets : BOOL;   // 1=New Oper valve cmd. resets fault, 0=reset req'd to clear fault
   Cfg_ShedOnFullStall : BOOL := 1;   // 1=Stop Valve and Alarm on Full Stall; 0=Alarm only on Full Stall
   Cfg_ShedOnTransitStall : BOOL := 1;   // 1=Stop Valve and Alarm on Transit Stall; 0=Alarm only on Transit Stall
   Cfg_ShedOnIOFault : BOOL := 1;   // 1=Stop Valve and Alarm on I/O Fault; 0=Alarm only on I/O Fault
   Cfg_OvrdPermIntlk : BOOL;   // 1=Override ignores Bypassable Perm/ Intlk; 0=always use Perm/Intlk
   Cfg_HasFullStallAlm : ALIAS FOR FullStall.Cfg_Exists;   // 1=Full Stall Alarm exists and will be checked
   Cfg_HasTransitStallAlm : ALIAS FOR TransitStall.Cfg_Exists;   // 1=Transit Stall Alarm exists and will be checked
   Cfg_HasIntlkTripAlm : ALIAS FOR IntlkTrip.Cfg_Exists;   // 1=Interlock Trip Alarm exists and will be checked
   Cfg_HasIOFaultAlm : ALIAS FOR IOFault.Cfg_Exists;   // 1=I/O Fault Alarm exists and will be checked
   Cfg_FullStallResetReqd : ALIAS FOR FullStall.Cfg_ResetReqd;   // 1=Reset requied to clear Full Stall Alarm
   Cfg_TransitStallResetReqd : ALIAS FOR TransitStall.Cfg_ResetReqd;   // 1=Reset required to clear Transit Stall Alarm
   Cfg_IntlkTripResetReqd : ALIAS FOR IntlkTrip.Cfg_ResetReqd;   // 1=Reset required to clear Interlock Trip Alarm
   Cfg_IOFaultResetReqd : ALIAS FOR IOFault.Cfg_ResetReqd;   // 1=Reset required to clear I/O Fault Alarm
   Cfg_FullStallAckReqd : ALIAS FOR FullStall.Cfg_AckReqd;   // 1=Acknowledge required for Full Stall Alarm
   Cfg_TransitStallAckReqd : ALIAS FOR TransitStall.Cfg_AckReqd;   // 1=Acknowledge required for Transit Stall Alarm
   Cfg_IntlkTripAckReqd : ALIAS FOR IntlkTrip.Cfg_AckReqd;   // 1=Acknowledge required for Interlock Trip Alarm
   Cfg_IOFaultAckReqd : ALIAS FOR IOFault.Cfg_AckReqd;   // 1=Acknowledge required for I/O Fault Alarm
   Cfg_FullStallSeverity : ALIAS FOR FullStall.Cfg_Severity;   // Full Stall Alarm Severity: 1..250=Low, 251..500=Medium, 501..750=High, 751..1000=Urgent
   Cfg_TransitStallSeverity : ALIAS FOR TransitStall.Cfg_Severity;   // Transit Stall Alarm Severity: 1..250=Low, 251..500=Medium, 501..750=High, 751..1000=Urgent
   Cfg_IntlkTripSeverity : ALIAS FOR IntlkTrip.Cfg_Severity;   // Interlock Trip Alarm Severity: 1..250=Low, 251..500=Medium, 501..750=High, 751..1000=Urgent
   Cfg_IOFaultSeverity : ALIAS FOR IOFault.Cfg_Severity;   // I/O Fault Alarm Severity: 1..250=Low, 251..500=Medium, 501..750=High, 751..1000=Urgent
   Cfg_SimFdbkT : DINT := 2;   // Delay to echo back of Open/Closed status when in Simulation (sec)
   Cfg_FullStallT : DINT := 5;   // After command, time with no motion before Fault (sec)
   Cfg_TransitStallT : DINT := 10;   // After command, time to reach position before fault (sec)
   PSet_Owner : DINT;   // Program Owner Request ID (non-zero) or Release (zero)
   PCmd_Open : BOOL;   // Program Command to Open Valve
   PCmd_Close : BOOL;   // Program Command to Close Valve
   PCmd_Acq : ALIAS FOR Mode.PCmd_Acq; {visible}
   PCmd_Rel : ALIAS FOR Mode.PCmd_Rel; {visible}
   PCmd_Lock : ALIAS FOR Mode.PCmd_Lock; {visible}
   PCmd_Unlock : ALIAS FOR Mode.PCmd_Unlock; {visible}
   PCmd_Reset : BOOL;   // Program Command to Reset all Alarms requiring Reset
   PCmd_FullStallAck : ALIAS FOR FullStall.PCmd_Ack;   // Program Command to Acknowledge Full Stall Alarm
   PCmd_FullStallSuppress : ALIAS FOR FullStall.PCmd_Suppress;   // Program Command to Suppress Full Stall Alarm
   PCmd_FullStallUnsuppress : ALIAS FOR FullStall.PCmd_Unsuppress;   // Program Command to Unsuppress Full Stall Alarm
   PCmd_FullStallUnshelve : ALIAS FOR FullStall.PCmd_Unshelve;   // Program Command to Unshelve Full Stall Alarm
   PCmd_TransitStallAck : ALIAS FOR TransitStall.PCmd_Ack;   // Program Command to Acknowledge Transit Stall Alarm
   PCmd_TransitStallSuppress : ALIAS FOR TransitStall.PCmd_Suppress;   // Program Command to Suppress Transit Stall Alarm
   PCmd_TransitStallUnsuppress : ALIAS FOR TransitStall.PCmd_Unsuppress;   // Program Command to Unsuppress Transit Stall Alarm
   PCmd_TransitStallUnshelve : ALIAS FOR TransitStall.PCmd_Unshelve;   // Program Command to Unshelve Transit Stall Alarm
   PCmd_IntlkTripAck : ALIAS FOR IntlkTrip.PCmd_Ack;   // Program Command to Acknowledge Interlock Trip Alarm
   PCmd_IntlkTripSuppress : ALIAS FOR IntlkTrip.PCmd_Suppress;   // Program Command to Suppress Interlock Trip Alarm
   PCmd_IntlkTripUnsuppress : ALIAS FOR IntlkTrip.PCmd_Unsuppress;   // Program Command to Unsuppress Interlock Trip Alarm
   PCmd_IntlkTripUnshelve : ALIAS FOR IntlkTrip.PCmd_Unshelve;   // Program Command to Unshelve Interlock Trip Alarm
   PCmd_IOFaultAck : ALIAS FOR IOFault.PCmd_Ack;   // Program Command to Acknowledge I/O Fault Alarm
   PCmd_IOFaultSuppress : ALIAS FOR IOFault.PCmd_Suppress;   // Program Command to Suppress I/O Fault Alarm
   PCmd_IOFaultUnsuppress : ALIAS FOR IOFault.PCmd_Unsuppress;   // Program Command to Unsuppress I/O Fault Alarm
   PCmd_IOFaultUnshelve : ALIAS FOR IOFault.PCmd_Unshelve;   // Program Command to Unshelve I/O Fault Alarm
   OCmd_Open : BOOL;   // Operator Command to Open Valve
   OCmd_Close : BOOL;   // Operator Command to Close Valve
   OCmd_Bypass : BOOL;   // Operator Command to Bypass all Bypassable Interlocks and Permissives
   OCmd_Check : BOOL;   // Operator Command to Check (not bypass) all Interlocks and Permissives
   MCmd_Disable : BOOL;   // Maintenance Command to Disable Valve
   MCmd_Enable : BOOL;   // Maintenance Command to Enable (allow to energize) Valve
   MCmd_Acq : ALIAS FOR Mode.MCmd_Acq;
   MCmd_Rel : ALIAS FOR Mode.MCmd_Rel;
   OCmd_AcqLock : ALIAS FOR Mode.OCmd_AcqLock;
   OCmd_Unlock : ALIAS FOR Mode.OCmd_UnlockRel;
   OCmd_Reset : BOOL;   // Operator Command to Reset all Alarms requiring Reset
   OCmd_ResetAckAll : BOOL;   // Operator Command to Reset all Alarms and latched Shed conditions
END_VAR
VAR_OUTPUT
   Out : BOOL; {access Read Only, visible}   // 1=Energize Valve Solenoid
   SrcQ_IO : DINT; {access Read Only}   // Source and Quality of primary I/O (enumeration)
   SrcQ : DINT; {access Read Only}   // Source and Quality of primary Val/Sts (enumeration)
   Val_Cmd : DINT; {access Read Only}   // Device Command 0=None, 1=Close, 2=Open
   Val_Fdbk : DINT; {access Read Only}   // Device Feedback 0=Moving, 1=Closed, 2=Opened, 3=Limit Switch Failure
   Val_Sts : DINT; {access Read Only}   // Device Confirmed Sts 0=? 1=Closed 2=Open 5=Closing, 6=Opening, 33=Disabled
   Val_Fault : DINT; {access Read Only}   // Device Fault Status 0=None, 16=Transit Stall, 17 = Full Stall, 32=I/O Fault, 34=Config Error
   Val_Mode : ALIAS FOR Mode.Val; {access Read Only}
   Val_Owner : DINT; {access Read Only}   // Current Object Owner ID (0=not owned)
   Val_Notify : DINT; {access Read Only}   // Current Alarm Level and Acknowledgement (enumeration)
   Sts_Closed : BOOL; {access Read Only, visible}   // 1=Valve requested to Close and is confirmed Closed
   Sts_Opening : BOOL; {access Read Only, visible}   // 1=Valve requested to open and awaiting open feedback
   Sts_Opened : BOOL; {access Read Only, visible}   // 1=Valve requested to open and is confirmed Opened
   Sts_Closing : BOOL; {access Read Only, visible}   // 1=Valve requested to Close and awaiting Closed feedback
   Sts_Available : BOOL; {access Read Only}   // 1=Valve available for control by automation (Prog)
   Sts_Bypass : BOOL; {access Read Only}   // 1=Bypassable Interlocks and Permissives are Bypassed
   Sts_BypActive : BOOL; {access Read Only}   // 1=Bypassing Active (Bypassed or Maintenance)
   Sts_Disabled : BOOL; {access Read Only}   // 1=Valve is Disabled
   Sts_LSFail : BOOL; {access Read Only}   // 1=Limit Switch Overlap Failure
   Sts_NotRdy : BOOL; {access Read Only}   // 1=Device Not Ready, see detail bits for reason
   Nrdy_Disabled : BOOL; {access Read Only}   // 1=Device Not Ready: Device Disabled by Maintenance
   Nrdy_CfgErr : BOOL; {access Read Only}   // 1=Device Not Ready: Configuration Error
   Nrdy_Intlk : BOOL; {access Read Only}   // 1=Device Not Ready: Interlock Not OK
   Nrdy_Perm : BOOL; {access Read Only}   // 1=Device Not Ready: Permissive Not OK
   Nrdy_Fail : BOOL; {access Read Only}   // 1=Device Not Ready: Device Failure (Shed Requires Reset)
   Nrdy_IOFault : BOOL; {access Read Only}   // 1=Device Not Ready: I/O Fault (Shed Requires Reset)
   Nrdy_NoMode : BOOL; {access Read Only}   // 1=Device Not Ready: Device Logic Disabled / NO Mode
   Sts_MaintByp : BOOL; {access Read Only}   // 1=A Maintenance Bypass is Active, display icon
   Sts_AlmInh : BOOL; {access Read Only}   // 1=An Alarm is Shelved, Disabled or Suppressed, display icon
   Sts_Err : BOOL; {access Read Only, visible}   // 1=Error in Config: see detail bits for reason
   Err_Timer : BOOL; {access Read Only}   // 1=Error in Config: Invalid Check Time (use 0 to 2147483)
   Err_Sim : BOOL; {access Read Only}   // 1=Error in Config: Invalid Simulation Time (use 0 to 2147483)
   Err_Alarm : BOOL; {access Read Only}   // 1=Error in Config: Alarm Min On Time, Shelf Time, Severity
   Sts_Hand : ALIAS FOR Mode.Sts_Hand; {access Read Only, visible}
   Sts_Maint : ALIAS FOR Mode.Sts_Maint; {access Read Only, visible}
   Sts_Ovrd : ALIAS FOR Mode.Sts_Ovrd; {access Read Only, visible}
   Sts_Prog : ALIAS FOR Mode.Sts_Prog; {access Read Only, visible}
   Sts_Oper : ALIAS FOR Mode.Sts_Oper; {access Read Only, visible}
   Sts_ProgOperLock : ALIAS FOR Mode.Sts_ProgOperLock; {access Read Only}
   Sts_NoMode : ALIAS FOR Mode.Sts_NoMode; {access Read Only}
   Sts_MAcqRcvd : ALIAS FOR Mode.Sts_MAcqRcvd; {access Read Only}
   Sts_FullStall : ALIAS FOR FullStall.Inp;   // 1=Valve Full Stall (failed to move at all)
   Alm_FullStall : ALIAS FOR FullStall.Alm;   // 1=Valve Full Stall (failed to move at all) Alarm
   Ack_FullStall : ALIAS FOR FullStall.Ack;   // 1=Full Stall Alarm has been acknowledged
   Sts_FullStallDisabled : ALIAS FOR FullStall.Disabled;   // 1=Full Stall Alarm has been Disabled by Maintenance
   Sts_FullStallShelved : ALIAS FOR FullStall.Shelved;   // 1=Full Stall Alarm has been Shelved by Operator
   Sts_FullStallSuppressed : ALIAS FOR FullStall.Suppressed;   // 1=Full Stall Alarm has been Suppressed by Program
   Sts_TransitStall : ALIAS FOR TransitStall.Inp;   // 1=Valve Transit Stall (did not reach target position)
   Alm_TransitStall : ALIAS FOR TransitStall.Alm;   // 1=Valve Transit Stall (did not reach target pos.) Alarm
   Ack_TransitStall : ALIAS FOR TransitStall.Ack;   // 1=Transit Stall Alarm has been acknowledged
   Sts_TransitStallDisabled : ALIAS FOR TransitStall.Disabled;   // 1=Transit Stall Alarm has been Disabled by Maintenance
   Sts_TransitStallShelved : ALIAS FOR TransitStall.Shelved;   // 1=Transit Stall Alarm has been Shelved by Operator
   Sts_TransitStallSuppressed : ALIAS FOR TransitStall.Suppressed;   // 1=Transit Stall Alarm has been Suppressed by Program
   Sts_IntlkTrip : ALIAS FOR IntlkTrip.Inp;   // 1=Valve de-energized by an Interlock NOT OK
   Alm_IntlkTrip : ALIAS FOR IntlkTrip.Alm;   // 1=Alarm: Valve de-energized by an Interlock NOT OK
   Ack_IntlkTrip : ALIAS FOR IntlkTrip.Ack;   // 1=Interlock Trip Alarm has been acknowledged
   Sts_IntlkTripDisabled : ALIAS FOR IntlkTrip.Disabled;   // 1=Interlock Trip Alarm has been Disabled by Maintenance
   Sts_IntlkTripShelved : ALIAS FOR IntlkTrip.Shelved;   // 1=Interlock Trip Alarm has been Shelved by Operator
   Sts_IntlkTripSuppressed : ALIAS FOR IntlkTrip.Suppressed;   // 1=Interlock Trip Alarm has been Suppressed Program
   Sts_IOFault : ALIAS FOR IOFault.Inp;   // I/O Comm Fault Status (0=OK, 1=Bad)
   Alm_IOFault : ALIAS FOR IOFault.Alm;   // 1=I/O Fault Alarm
   Ack_IOFault : ALIAS FOR IOFault.Ack;   // 1=I/O Fault Alarm has been acknowledged
   Sts_IOFaultDisabled : ALIAS FOR IOFault.Disabled;   // 1=I/O Fault Alarm has been Disabled by Maintenance
   Sts_IOFaultShelved : ALIAS FOR IOFault.Shelved;   // 1=I/O Fault Alarm has been Shelved by Operator
   Sts_IOFaultSuppressed : ALIAS FOR IOFault.Suppressed;   // 1=I/O Fault Alarm has been Suppressed by Program
   Rdy_Open : BOOL; {access Read Only}   // 1=Ready to receive OCmd_Open (enables HMI button)
   Rdy_Close : BOOL; {access Read Only}   // 1=Ready to receive OCmd_Close (enables HMI button)
   Rdy_Bypass : BOOL; {access Read Only}   // 1=Ready to receive OCmd_Bypass (enables HMI button)
   Rdy_Check : BOOL; {access Read Only}   // 1=Ready to receive OCmd_Check (enables HMI button)
   Rdy_Disable : BOOL; {access Read Only}   // 1=Ready to receive MCmd_Disable (enables HMI button)
   Rdy_Enable : BOOL; {access Read Only}   // 1=Ready to receive MCmd_Enable (enables HMI button)
   Rdy_Reset : BOOL; {access Read Only}   // 1=Ready to receive OCmd_Reset (enables HMI button)
   Rdy_ResetAckAll : BOOL; {access Read Only}   // 1=At least one Alarm or latched Shed condition requires Reset or Ack
   P_ValveSO : BOOL;   // Unique Parameter Name for auto - discovery
END_VAR
VAR_INPUT
   HMI_OvrdCmd : DINT;   // HMI Ovrd command 1 = Close 2 = Open
END_VAR
VAR
   Mode : P_Mode := (Cfg_OvrdOverLock := 1, Rdy_OAcq := 1);   // Valve Mode Selection
   IOFault : P_Alarm := (Cfg_AckReqd := 1, Cfg_AllowShelve := 1, Cfg_AllowDisable := 1, Cfg_PCmdClear := 1, Cfg_Severity := 1000, Cfg_AlmMinOnT := 5, PCfg_AllowExist := 1, Ack := 1);   // I/O Fault Alarm
   IntlkTrip : P_Alarm := (Cfg_AckReqd := 1, Cfg_AllowShelve := 1, Cfg_AllowDisable := 1, Cfg_PCmdClear := 1, Cfg_Severity := 500, Cfg_AlmMinOnT := 5, PCfg_AllowExist := 1, Ack := 1);   // Interlock Trip Alarm
   TransitStall : P_Alarm := (Cfg_AckReqd := 1, Cfg_AllowShelve := 1, Cfg_AllowDisable := 1, Cfg_PCmdClear := 1, Cfg_Severity := 1000, Cfg_AlmMinOnT := 5, PCfg_AllowExist := 1, Ack := 1);   // Valve Transit Stall (moved but did not reach target) Alarm
   FullStall : P_Alarm := (Cfg_AckReqd := 1, Cfg_AllowShelve := 1, Cfg_AllowDisable := 1, Cfg_PCmdClear := 1, Cfg_Severity := 1000, Cfg_AlmMinOnT := 5, PCfg_AllowExist := 1, Ack := 1);   // Valve Full Stall (did not move) Alarm
   Cfg_Tag : STRING_12;   // Tagname for display on HMI
   Wrk_Open : BOOL; {access None}   // 1=Requested to OPEN Valve, 0=Requested to CLOSE Valve
   Wrk_SimOpenT : TIMER; {access None}   // Simulation Delay until Opened
   Wrk_SimCloseT : TIMER; {access None}   // Simulation Delay until Closed
   Wrk_OpenFdbk : BOOL; {access None}   // 1=LS Feedback shows valve confirmed open
   Wrk_Notify : DINT; {access None}   // Buffer for building Val_Notify
   Wrk_Bypass : BOOL; {access None}   // Internal Bypassable Permissives and Interlocks are Bypassed flag
   Wrk_Disabled : BOOL; {access None}   // Internal Valve is Disabled
   Wrk_ClosedFdbk : BOOL; {access None}   // 1=LS Feedback shows valve confirmed closed
   Wrk_TransitStallT : TIMER; {access Read Only}   // Timer for Transit Stall Check
   Wrk_FullStallT : TIMER; {access Read Only}   // Timer for Full Stall Check
   Inf_Tab : DINT;   // Tab to display (FTView ME)
   Wrk_Sts : DINT; {access None}   // Buffer for building Val_Sts
   Wrk_SrcQ : DINT; {access None}   // Register for building Source / Quality enumeration
   Wrk_Fault : DINT; {access None}   // Buffer for building Val_Fault
   Wrk_Cmd : DINT; {access None}   // Buffer for building Val_Cmd
   Wrk_SimOpenLS : BOOL; {access None}   // Simulated valve Open Limit Switch
   Wrk_SimClosedLS : BOOL; {access None}   // Simulated valve Closed Limit Switch
   Wrk_NotRdy : BOOL; {access None}   // Device Not Ready conditions excluding shed latches
   Wrk_NoLongerSim : BOOL; {access None}   // Switched from Simulated to Real Valve this scan
END_VAR

ROUTINE EnableInFalse   (* ladder *)
// Disabled is asserted; Outputs OFF; Valve Status shown but Alarms disabled
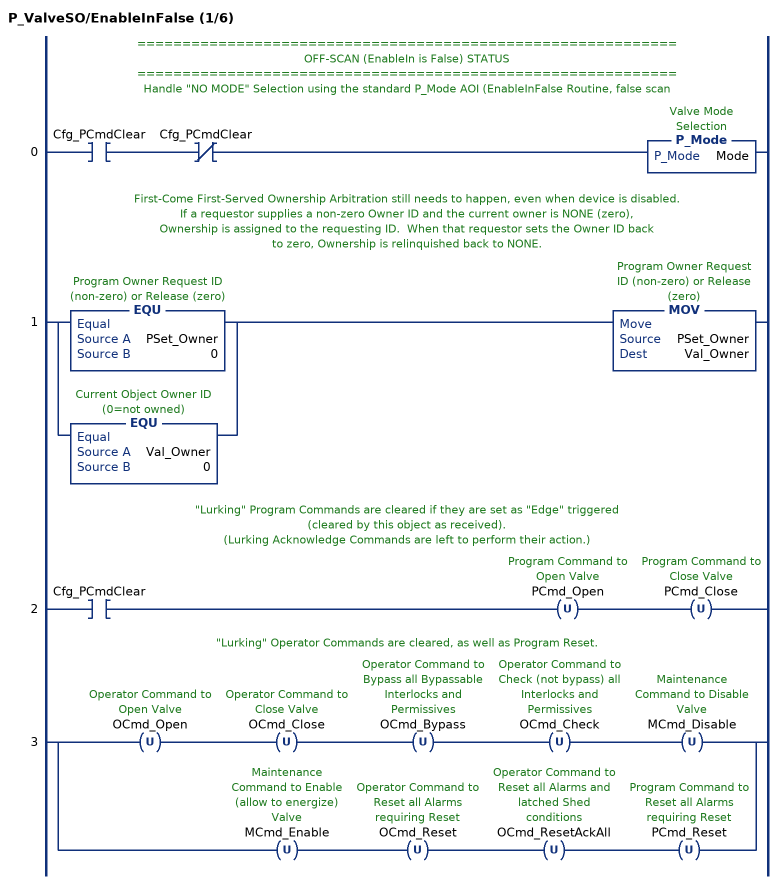
   // ============================================================
   // OFF-SCAN (EnableIn is False) STATUS
   // ============================================================
   // Handle "NO MODE" Selection using the standard P_Mode AOI (EnableInFalse Routine, false scan
   0: XIC(Cfg_PCmdClear)XIO(Cfg_PCmdClear)P_Mode(Mode);
   // First-Come First-Served Ownership Arbitration still needs to happen, even when device is disabled.
   // If a requestor supplies a non-zero Owner ID and the current owner is NONE (zero),
   // Ownership is assigned to the requesting ID.  When that requestor sets the Owner ID back
   // to zero, Ownership is relinquished back to NONE.
   1: [EQU(PSet_Owner,0) ,EQU(Val_Owner,0) ]MOV(PSet_Owner,Val_Owner);
   // "Lurking" Program Commands are cleared if they are set as "Edge" triggered
   // (cleared by this object as received).
   // (Lurking Acknowledge Commands are left to perform their action.)
   2: XIC(Cfg_PCmdClear)OTU(PCmd_Open)OTU(PCmd_Close);
   // "Lurking" Operator Commands are cleared, as well as Program Reset.
   3: [OTU(OCmd_Open) OTU(OCmd_Close) OTU(OCmd_Bypass) OTU(OCmd_Check) OTU(MCmd_Disable) ,OTU(MCmd_Enable) OTU(OCmd_Reset) OTU(OCmd_ResetAckAll) OTU(PCmd_Reset) ];
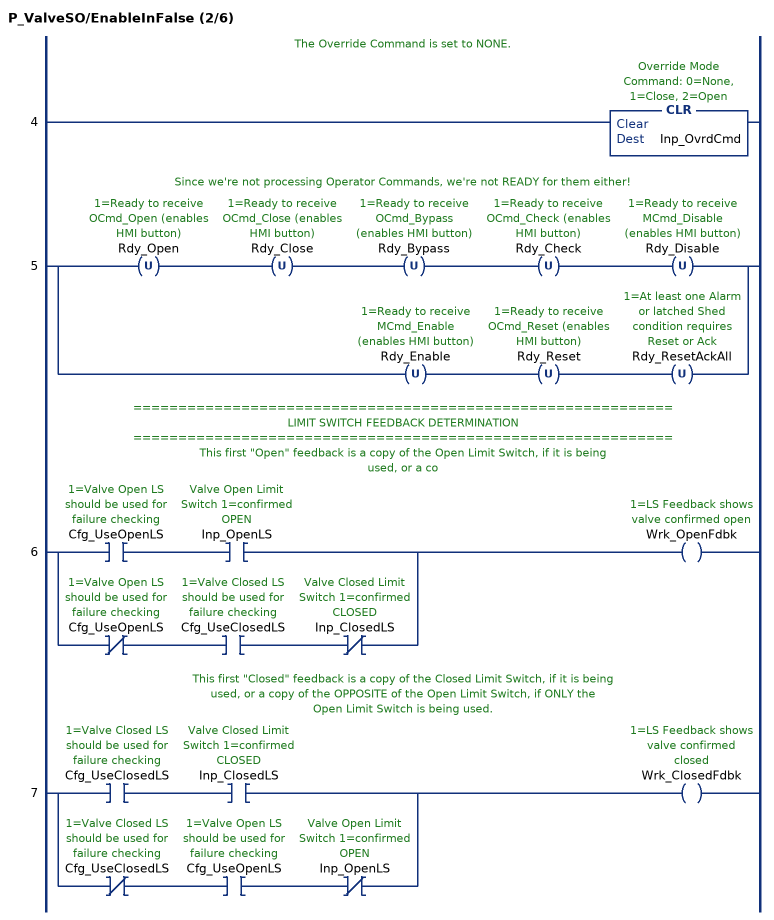
   // The Override Command is set to NONE.
   4: CLR(Inp_OvrdCmd);
   // Since we're not processing Operator Commands, we're not READY for them either!
   5: [OTU(Rdy_Open) OTU(Rdy_Close) OTU(Rdy_Bypass) OTU(Rdy_Check) OTU(Rdy_Disable) ,OTU(Rdy_Enable) OTU(Rdy_Reset) OTU(Rdy_ResetAckAll) ];
   // ============================================================
   // LIMIT SWITCH FEEDBACK DETERMINATION
   // ============================================================
   // This first "Open" feedback is a copy of the Open Limit Switch, if it is being
   // used, or a co
   6: [XIC(Cfg_UseOpenLS) XIC(Inp_OpenLS) ,XIO(Cfg_UseOpenLS) XIC(Cfg_UseClosedLS) XIO(Inp_ClosedLS) ]OTE(Wrk_OpenFdbk);
   // This first "Closed" feedback is a copy of the Closed Limit Switch, if it is being
   // used, or a copy of the OPPOSITE of the Open Limit Switch, if ONLY the
   // Open Limit Switch is being used.
   7: [XIC(Cfg_UseClosedLS) XIC(Inp_ClosedLS) ,XIO(Cfg_UseClosedLS) XIC(Cfg_UseOpenLS) XIO(Inp_OpenLS) ]OTE(Wrk_ClosedFdbk);
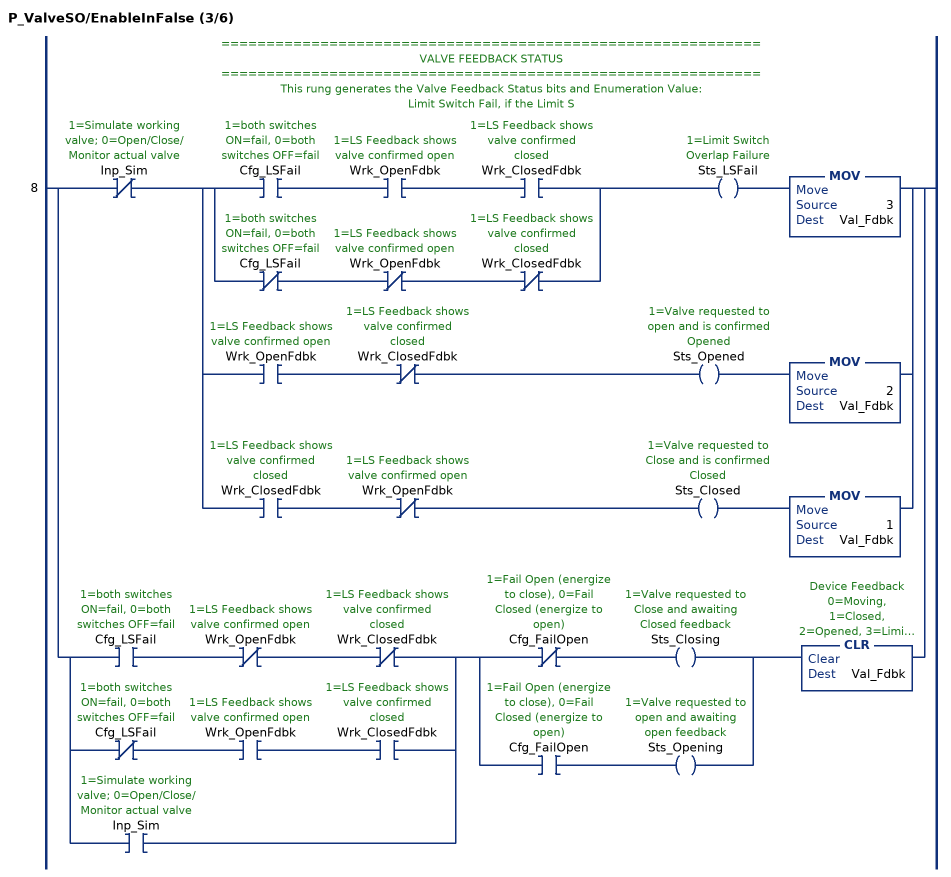
   // ============================================================
   // VALVE FEEDBACK STATUS
   // ============================================================
   // This rung generates the Valve Feedback Status bits and Enumeration Value:
   // Limit Switch Fail, if the Limit S
   8: [XIO(Inp_Sim) [[XIC(Cfg_LSFail) XIC(Wrk_OpenFdbk) XIC(Wrk_ClosedFdbk) ,XIO(Cfg_LSFail) XIO(Wrk_OpenFdbk) XIO(Wrk_ClosedFdbk) ] OTE(Sts_LSFail) MOV(3,Val_Fdbk) ,XIC(Wrk_OpenFdbk) XIO(Wrk_ClosedFdbk) OTE(Sts_Opened) MOV(2,Val_Fdbk) ,XIC(Wrk_ClosedFdbk) XIO(Wrk_OpenFdbk) OTE(Sts_Closed) MOV(1,Val_Fdbk) ] ,[[XIC(Cfg_LSFail) XIO(Wrk_OpenFdbk) XIO(Wrk_ClosedFdbk) ,XIO(Cfg_LSFail) XIC(Wrk_OpenFdbk) XIC(Wrk_ClosedFdbk) ] ,XIC(Inp_Sim) ] [XIO(Cfg_FailOpen) OTE(Sts_Closing) ,XIC(Cfg_FailOpen) OTE(Sts_Opening) ] CLR(Val_Fdbk) ];
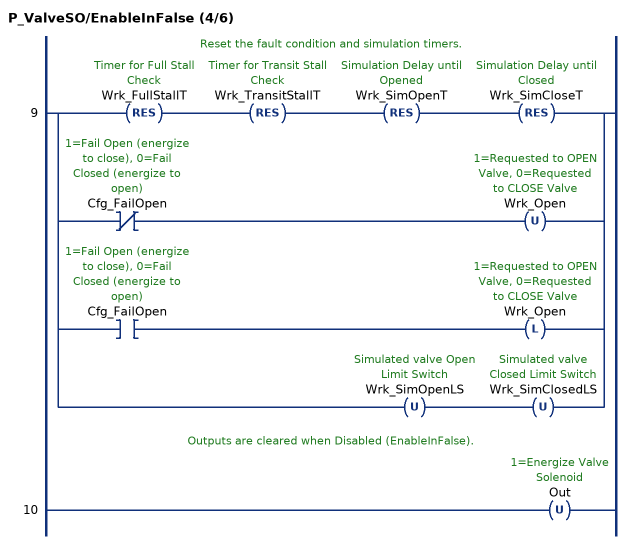
   // Reset the fault condition and simulation timers.
   9: [RES(Wrk_FullStallT) RES(Wrk_TransitStallT) RES(Wrk_SimOpenT) RES(Wrk_SimCloseT) ,[XIO(Cfg_FailOpen) OTU(Wrk_Open) ,XIC(Cfg_FailOpen) OTL(Wrk_Open) ] ,OTU(Wrk_SimOpenLS) OTU(Wrk_SimClosedLS) ];
   // Outputs are cleared when Disabled (EnableInFalse).
   10: OTU(Out);
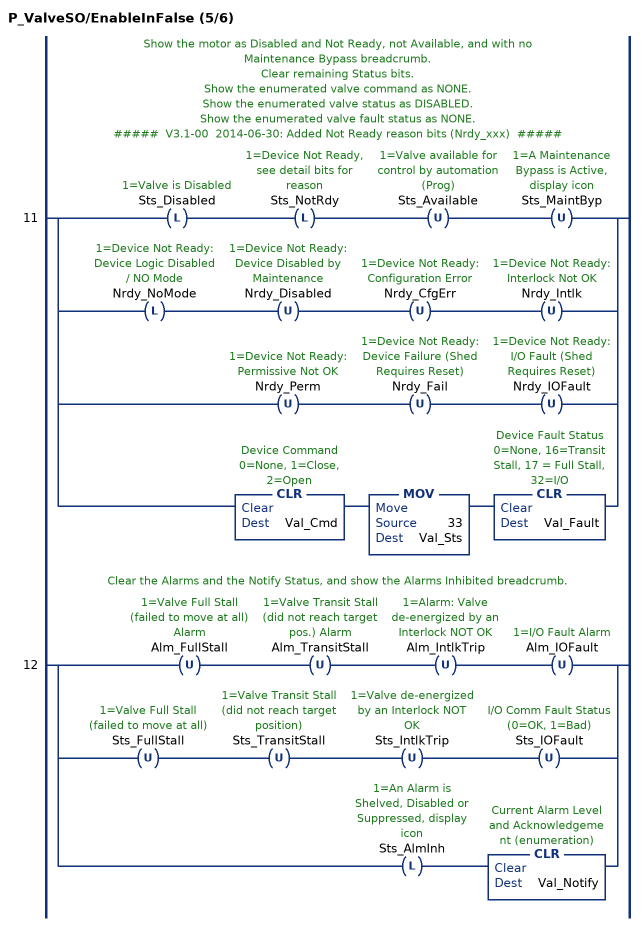
   // Show the motor as Disabled and Not Ready, not Available, and with no
   // Maintenance Bypass breadcrumb.
   // Clear remaining Status bits.
   // Show the enumerated valve command as NONE.
   // Show the enumerated valve status as DISABLED.
   // Show the enumerated valve fault status as NONE.
   // #####  V3.1-00  2014-06-30: Added Not Ready reason bits (Nrdy_xxx)  #####
   11: [OTL(Sts_Disabled) OTL(Sts_NotRdy) OTU(Sts_Available) OTU(Sts_MaintByp) ,OTL(Nrdy_NoMode) OTU(Nrdy_Disabled) OTU(Nrdy_CfgErr) OTU(Nrdy_Intlk) ,OTU(Nrdy_Perm) OTU(Nrdy_Fail) OTU(Nrdy_IOFault) ,CLR(Val_Cmd) MOV(33,Val_Sts) CLR(Val_Fault) ];
   // Clear the Alarms and the Notify Status, and show the Alarms Inhibited breadcrumb.
   12: [OTU(Alm_FullStall) OTU(Alm_TransitStall) OTU(Alm_IntlkTrip) OTU(Alm_IOFault) ,OTU(Sts_FullStall) OTU(Sts_TransitStall) OTU(Sts_IntlkTrip) OTU(Sts_IOFault) ,OTL(Sts_AlmInh) CLR(Val_Notify) ];
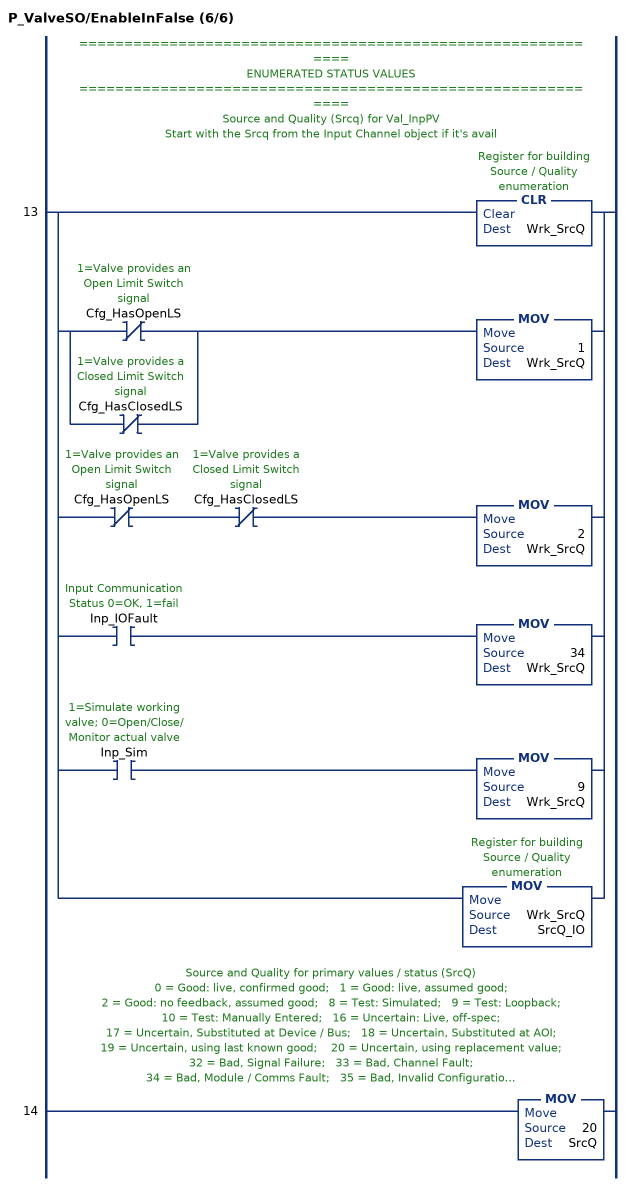
   // ============================================================
   // ENUMERATED STATUS VALUES
   // ============================================================
   // Source and Quality (Srcq) for Val_InpPV
   // Start with the Srcq from the Input Channel object if it's avail
   13: [CLR(Wrk_SrcQ) ,[XIO(Cfg_HasOpenLS) ,XIO(Cfg_HasClosedLS) ] MOV(1,Wrk_SrcQ) ,XIO(Cfg_HasOpenLS) XIO(Cfg_HasClosedLS) MOV(2,Wrk_SrcQ) ,XIC(Inp_IOFault) MOV(34,Wrk_SrcQ) ,XIC(Inp_Sim) MOV(9,Wrk_SrcQ) ,MOV(Wrk_SrcQ,SrcQ_IO) ];
   // Source and Quality for primary values / status (SrcQ)
   // 0 = Good: live, confirmed good;   1 = Good: live, assumed good;
   // 2 = Good: no feedback, assumed good;   8 = Test: Simulated;   9 = Test: Loopback;
   // 10 = Test: Manually Entered;   16 = Uncertain: Live, off-spec;
   // 17 = Uncertain, Substituted at Device / Bus;   18 = Uncertain, Substituted at AOI;
   // 19 = Uncertain, using last known good;    20 = Uncertain, using replacement value;
   // 32 = Bad, Signal Failure;   33 = Bad, Channel Fault;
   // 34 = Bad, Module / Comms Fault;   35 = Bad, Invalid Configuration
   // #####  V3.1-00  2014-06-30:  Added rung for Source/Quality enumerations.  #####
   14: MOV(20,SrcQ);
END_ROUTINE
